KUKA KRL program: MyProgram_126().src

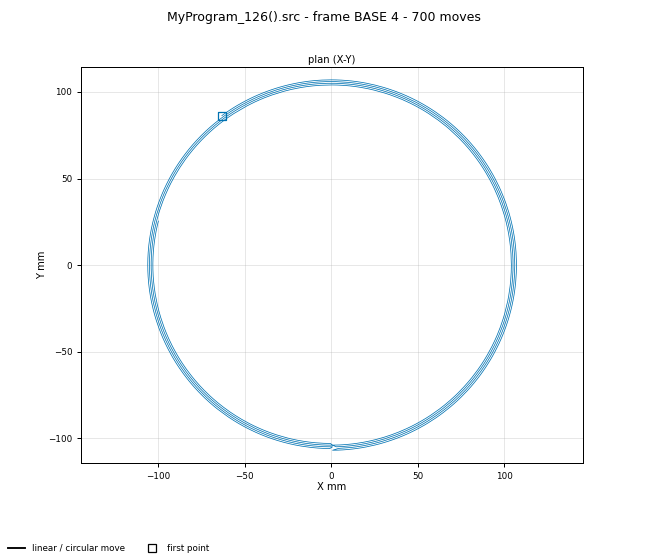
[picture p0: tool path of MyProgram_126().src in frame BASE 4, 700 of 700 moves have a stored position in this frame; points joined in program order, loops and branches not executed]
&ACCESS RVP
&REL 1
&PARAM TEMPLATE = C:\KRC\Roboter\Template\vorgabe
&PARAM EDITMASK = *
DEF MyProgram_126()
; ---- Setting reference (Base) ----
$BASE = BASE_DATA[4]

; --------------------------
; ---- Setting tool (TCP) ----
$TOOL = TOOL_DATA[3]
; --------------------------

$VEL.CP = VEL_APROX_PRINT
Startdeposition()
$VEL.CP = VEL_PRINT
LIN {X -63.1744,Y 86.354,Z 105,A 121.2635,B 24.9294,C -1.9405,E1 24.9063,E2 324.4003} C_DIS
LIN {X -61.0361,Y 87.8784,Z 105,A 119.8304,B 24.9293,C -1.9424,E1 24.9096,E2 325.8339} C_DIS
LIN {X -58.6968,Y 89.4582,Z 105,A 118.2628,B 24.9293,C -1.9432,E1 24.9133,E2 327.4047} C_DIS
LIN {X -56.1298,Y 91.0928,Z 105,A 116.6759,B 24.9289,C -1.9479,E1 24.917,E2 328.9856} C_DIS
LIN {X -53.8773,Y 92.4429,Z 105,A 115.2641,B 24.9287,C -1.9502,E1 24.9204,E2 330.3961} C_DIS
LIN {X -51.5924,Y 93.7373,Z 105,A 113.8527,B 24.9285,C -1.9525,E1 24.9238,E2 331.8062} C_DIS
LIN {X -49.2765,Y 94.9752,Z 105,A 112.4412,B 24.9284,C -1.9546,E1 24.9273,E2 333.2165} C_DIS
LIN {X -46.9308,Y 96.1559,Z 105,A 111.03,B 24.9282,C -1.9567,E1 24.9308,E2 334.6265} C_DIS
LIN {X -44.5569,Y 97.2787,Z 105,A 109.6191,B 24.9281,C -1.9587,E1 24.9344,E2 336.0362} C_DIS
LIN {X -42.1561,Y 98.3428,Z 105,A 108.2082,B 24.9279,C -1.9606,E1 24.938,E2 337.4459} C_DIS
LIN {X -39.73,Y 99.3478,Z 105,A 106.7979,B 24.9278,C -1.9624,E1 24.9416,E2 338.8551} C_DIS
LIN {X -37.2799,Y 100.2929,Z 105,A 105.3874,B 24.9277,C -1.9641,E1 24.9453,E2 340.2644} C_DIS
LIN {X -34.8074,Y 101.1776,Z 105,A 103.9775,B 24.9276,C -1.9657,E1 24.949,E2 341.6733} C_DIS
LIN {X -32.3139,Y 102.0013,Z 105,A 102.5675,B 24.9274,C -1.9672,E1 24.9528,E2 343.0822} C_DIS
LIN {X -29.8009,Y 102.7636,Z 105,A 101.1579,B 24.9274,C -1.9687,E1 24.9566,E2 344.4908} C_DIS
LIN {X -27.27,Y 103.464,Z 105,A 99.7486,B 24.9272,C -1.97,E1 24.9604,E2 345.8991} C_DIS
LIN {X -24.7226,Y 104.1021,Z 105,A 98.1893,B 24.9276,C -1.9655,E1 24.9646,E2 347.4712} C_DIS
LIN {X -21.4758,Y 104.818,Z 105,A 96.576,B 24.927,C -1.9735,E1 24.969,E2 349.0675} C_DIS
LIN {X -18.7569,Y 105.3387,Z 105,A 95.0092,B 24.9271,C -1.9714,E1 24.9733,E2 350.6409} C_DIS
LIN {X -15.6998,Y 105.8394,Z 105,A 93.4091,B 24.9269,C -1.9748,E1 24.9777,E2 352.2345} C_DIS
LIN {X -13.0976,Y 106.1928,Z 105,A 92.001,B 24.9269,C -1.9755,E1 24.9816,E2 353.6417} C_DIS
LIN {X -10.4876,Y 106.4822,Z 105,A 90.5932,B 24.9268,C -1.9762,E1 24.9855,E2 355.0487} C_DIS
LIN {X -7.8712,Y 106.7075,Z 105,A 89.1853,B 24.9268,C -1.9768,E1 24.9894,E2 356.4559} C_DIS
LIN {X -5.2501,Y 106.8686,Z 105,A 87.778,B 24.9267,C -1.9773,E1 24.9933,E2 357.8624} C_DIS
LIN {X -2.6258,Y 106.9652,Z 105,A 86.3708,B 24.9267,C -1.9777,E1 24.9973,E2 359.2689} C_DIS
LIN {X -0.0646,Y 106.9971,Z 105,A 84.9971,B 24.9267,C -1.9779,E1 25.0011,E2 360.6421} C_DIS
LIN {X 2.7297,Y 106.962,Z 105,A 83.3358,B 24.9271,C -1.9716,E1 25.0058,E2 362.318} C_DIS
LIN {X 5.8633,Y 106.8347,Z 105,A 81.8013,B 24.9267,C -1.9774,E1 25.01,E2 363.8383} C_DIS
LIN {X 8.8815,Y 106.6268,Z 105,A 80.1746,B 24.9267,C -1.9771,E1 25.0145,E2 365.465} C_DIS
LIN {X 11.7935,Y 106.3455,Z 105,A 78.6358,B 24.9267,C -1.9779,E1 25.0188,E2 367.0008} C_DIS
LIN {X 14.8232,Y 105.9639,Z 105,A 76.9473,B 24.9268,C -1.9755,E1 25.0235,E2 368.6937} C_DIS
LIN {X 17.6867,Y 105.5235,Z 105,A 75.4509,B 24.9268,C -1.9772,E1 25.0276,E2 370.1846} C_DIS
LIN {X 20.2711,Y 105.0576,Z 105,A 74.0666,B 24.9267,C -1.9775,E1 25.0314,E2 371.5666} C_DIS
LIN {X 22.8432,Y 104.5285,Z 105,A 72.6618,B 24.9267,C -1.9769,E1 25.0352,E2 372.9711} C_DIS
LIN {X 25.3193,Y 103.9565,Z 105,A 71.2816,B 24.9268,C -1.9753,E1 25.039,E2 374.3529} C_DIS
LIN {X 27.9447,Y 103.2818,Z 105,A 69.8529,B 24.9268,C -1.9753,E1 25.0428,E2 375.7794} C_DIS
LIN {X 30.3725,Y 102.594,Z 105,A 68.4576,B 24.927,C -1.9726,E1 25.0466,E2 377.1788} C_DIS
LIN {X 32.9788,Y 101.7862,Z 105,A 67.0452,B 24.927,C -1.9734,E1 25.0504,E2 378.5867} C_DIS
LIN {X 35.4669,Y 100.9462,Z 105,A 65.6414,B 24.927,C -1.9723,E1 25.0541,E2 379.9903} C_DIS
LIN {X 37.9335,Y 100.0454,Z 105,A 64.2171,B 24.9272,C -1.9702,E1 25.0578,E2 381.4165} C_DIS
LIN {X 40.7094,Y 98.9491,Z 105,A 62.6093,B 24.9274,C -1.9682,E1 25.062,E2 383.0255} C_DIS
LIN {X 43.3598,Y 97.8181,Z 105,A 61.0832,B 24.9274,C -1.9672,E1 25.0659,E2 384.5504} C_DIS
LIN {X 45.7473,Y 96.7246,Z 105,A 59.6806,B 24.9276,C -1.9656,E1 25.0694,E2 385.953} C_DIS
LIN {X 48.5601,Y 95.3413,Z 105,A 57.9774,B 24.9278,C -1.9625,E1 25.0737,E2 387.6589} C_DIS
LIN {X 50.9781,Y 94.0705,Z 105,A 56.5274,B 24.9278,C -1.9611,E1 25.0773,E2 389.1083} C_DIS
LIN {X 53.3448,Y 92.7489,Z 105,A 55.1011,B 24.928,C -1.9601,E1 25.0807,E2 390.5327} C_DIS
LIN {X 55.9034,Y 91.2304,Z 105,A 53.5,B 24.9282,C -1.9574,E1 25.0845,E2 392.1353} C_DIS
LIN {X 58.3484,Y 89.6879,Z 105,A 51.97,B 24.9282,C -1.9556,E1 25.0881,E2 393.6644} C_DIS
LIN {X 60.5319,Y 88.229,Z 105,A 50.5686,B 24.9285,C -1.9535,E1 25.0914,E2 395.0661} C_DIS
LIN {X 62.6789,Y 86.7169,Z 105,A 49.1677,B 24.9286,C -1.9513,E1 25.0946,E2 396.4672} C_DIS
LIN {X 64.7784,Y 85.1599,Z 105,A 47.7733,B 24.9288,C -1.9491,E1 25.0977,E2 397.862} C_DIS
LIN {X 66.8584,Y 83.5369,Z 105,A 46.3663,B 24.929,C -1.9467,E1 25.1008,E2 399.2694} C_DIS
LIN {X 68.8883,Y 81.871,Z 105,A 44.9655,B 24.9291,C -1.9442,E1 25.1038,E2 400.6706} C_DIS
LIN {X 70.8768,Y 80.1557,Z 105,A 43.5655,B 24.9293,C -1.9417,E1 25.1067,E2 402.071} C_DIS
LIN {X 72.8226,Y 78.3921,Z 105,A 42.1654,B 24.9295,C -1.9391,E1 25.1096,E2 403.4717} C_DIS
LIN {X 74.7245,Y 76.5814,Z 105,A 40.7655,B 24.9297,C -1.9364,E1 25.1124,E2 404.872} C_DIS
LIN {X 76.5814,Y 74.7245,Z 105,A 39.3658,B 24.9299,C -1.9337,E1 25.1152,E2 406.2723} C_DIS
LIN {X 78.3921,Y 72.8226,Z 105,A 37.8771,B 24.9304,C -1.9271,E1 25.118,E2 407.77} C_DIS
LIN {X 80.5597,Y 70.4142,Z 105,A 36.1898,B 24.9305,C -1.9252,E1 25.1212,E2 409.4543} C_DIS
LIN {X 82.7102,Y 67.8785,Z 105,A 34.4682,B 24.9306,C -1.9234,E1 25.1242,E2 411.1721} C_DIS
LIN {X 84.3511,Y 65.8282,Z 105,A 33.0692,B 24.9309,C -1.9203,E1 25.1267,E2 412.5719} C_DIS
LIN {X 85.9412,Y 63.7383,Z 105,A 31.6706,B 24.9311,C -1.9172,E1 25.129,E2 413.9712} C_DIS
LIN {X 87.4795,Y 61.61,Z 105,A 30.2719,B 24.9313,C -1.914,E1 25.1313,E2 415.3707} C_DIS
LIN {X 88.9651,Y 59.4446,Z 105,A 28.8735,B 24.9316,C -1.9107,E1 25.1335,E2 416.7699} C_DIS
LIN {X 90.3972,Y 57.2434,Z 105,A 27.475,B 24.9318,C -1.9074,E1 25.1356,E2 418.1692} C_DIS
LIN {X 91.7748,Y 55.0077,Z 105,A 25.9012,B 24.9326,C -1.8965,E1 25.1379,E2 419.7607} C_DIS
LIN {X 93.4378,Y 52.1286,Z 105,A 24.3272,B 24.9323,C -1.9005,E1 25.14,E2 421.3171} C_DIS
LIN {X 94.689,Y 49.8199,Z 105,A 22.9293,B 24.9325,C -1.897,E1 25.1419,E2 422.7159} C_DIS
LIN {X 95.8831,Y 47.4811,Z 105,A 21.5111,B 24.9329,C -1.8925,E1 25.1437,E2 424.1371} C_DIS
LIN {X 96.9837,Y 45.1905,Z 105,A 20.138,B 24.9332,C -1.8882,E1 25.1453,E2 425.5132} C_DIS
LIN {X 98.0974,Y 42.7191,Z 105,A 18.7158,B 24.9334,C -1.8852,E1 25.1469,E2 426.9345} C_DIS
LIN {X 99.1163,Y 40.2988,Z 105,A 17.3391,B 24.9336,C -1.8824,E1 25.1484,E2 428.3102} C_DIS
LIN {X 100.0454,Y 37.9335,Z 105,A 15.9456,B 24.934,C -1.877,E1 25.1498,E2 429.7088} C_DIS
LIN {X 100.9462,Y 35.4668,Z 105,A 14.5483,B 24.9342,C -1.8732,E1 25.1511,E2 431.1072} C_DIS
LIN {X 101.8123,Y 32.8982,Z 105,A 13.1473,B 24.9344,C -1.871,E1 25.1523,E2 432.5055} C_DIS
LIN {X 102.5649,Y 30.4709,Z 105,A 11.7541,B 24.9348,C -1.8655,E1 25.1535,E2 433.9037} C_DIS
LIN {X 103.2818,Y 27.9447,Z 105,A 10.357,B 24.935,C -1.8616,E1 25.1545,E2 435.302} C_DIS
LIN {X 103.9859,Y 25.199,Z 105,A 8.8143,B 24.9354,C -1.8558,E1 25.1556,E2 436.8494} C_DIS
LIN {X 104.6775,Y 22.1604,Z 105,A 7.2123,B 24.9356,C -1.8535,E1 25.1565,E2 438.4476} C_DIS
LIN {X 105.1898,Y 19.5848,Z 105,A 5.8156,B 24.9359,C -1.8495,E1 25.1573,E2 439.8456} C_DIS
LIN {X 105.696,Y 16.627,Z 105,A 4.1294,B 24.9365,C -1.841,E1 25.158,E2 441.5418} C_DIS
LIN {X 106.1237,Y 13.6311,Z 105,A 2.534,B 24.9367,C -1.8369,E1 25.1586,E2 443.1374} C_DIS
LIN {X 106.4822,Y 10.4876,Z 105,A 0.9274,B 24.9369,C -1.8353,E1 25.1591,E2 444.7384} C_DIS
LIN {X 106.7394,Y 7.4006,Z 105,A -0.7805,B 24.9374,C -1.8279,E1 25.1595,E2 446.4537} C_DIS
LIN {X 106.8986,Y 4.5519,Z 105,A -2.2374,B 24.9375,C -1.826,E1 25.1597,E2 447.9063} C_DIS
LIN {X 106.9765,Y 2.0118,Z 105,A -3.6153,B 24.9379,C -1.8209,E1 25.1597,E2 449.2881} C_DIS
LIN {X 106.9894,Y -1.313,Z 105,A -5.3568,B 24.9381,C -1.8168,E1 25.1597,E2 451.029} C_DIS
LIN {X 106.8986,Y -4.5519,Z 105,A -7.0801,B 24.9385,C -1.8117,E1 25.1596,E2 452.754} C_DIS
LIN {X 106.749,Y -7.2585,Z 105,A -8.5008,B 24.9387,C -1.8083,E1 25.1594,E2 454.1742} C_DIS
LIN {X 106.5465,Y -9.7916,Z 105,A -9.8935,B 24.9391,C -1.8025,E1 25.159,E2 455.5723} C_DIS
LIN {X 106.2741,Y -12.4035,Z 105,A -11.2899,B 24.9394,C -1.7984,E1 25.1586,E2 456.9701} C_DIS
LIN {X 105.9377,Y -15.0078,Z 105,A -12.6659,B 24.9396,C -1.7951,E1 25.1581,E2 458.3457} C_DIS
LIN {X 105.5375,Y -17.6032,Z 105,A -14.0828,B 24.9399,C -1.7901,E1 25.1575,E2 459.766} C_DIS
LIN {X 104.993,Y -20.6067,Z 105,A -15.7082,B 24.9403,C -1.7853,E1 25.1566,E2 461.3934} C_DIS
LIN {X 104.3976,Y -23.4433,Z 105,A -17.2269,B 24.9405,C -1.7817,E1 25.1557,E2 462.9117} C_DIS
LIN {X 103.7909,Y -25.9983,Z 105,A -18.8086,B 24.9413,C -1.7696,E1 25.1546,E2 464.5128} C_DIS
LIN {X 102.9542,Y -29.1285,Z 105,A -20.3672,B 24.9412,C -1.7718,E1 25.1535,E2 466.0574} C_DIS
LIN {X 102.2083,Y -31.6463,Z 105,A -21.764,B 24.9414,C -1.7677,E1 25.1524,E2 467.4557} C_DIS
LIN {X 101.2929,Y -34.4655,Z 105,A -23.3577,B 24.9418,C -1.7624,E1 25.151,E2 469.0529} C_DIS
LIN {X 100.2929,Y -37.2799,Z 105,A -24.9085,B 24.942,C -1.7595,E1 25.1495,E2 470.6019} C_DIS
LIN {X 99.3478,Y -39.73,Z 105,A -26.3054,B 24.9422,C -1.7556,E1 25.1481,E2 472.0003} C_DIS
LIN {X 98.2923,Y -42.2721,Z 105,A -27.9259,B 24.9429,C -1.7448,E1 25.1463,E2 473.6375} C_DIS
LIN {X 96.9837,Y -45.1905,Z 105,A -29.4507,B 24.9428,C -1.7477,E1 25.1445,E2 475.1471} C_DIS
LIN {X 95.8831,Y -47.4811,Z 105,A -30.8236,B 24.9431,C -1.7431,E1 25.1428,E2 476.5235} C_DIS
LIN {X 94.689,Y -49.8199,Z 105,A -32.2941,B 24.9435,C -1.7361,E1 25.1409,E2 478.0027} C_DIS
LIN {X 93.0971,Y -52.7389,Z 105,A -33.9899,B 24.9436,C -1.7345,E1 25.1387,E2 479.6934} C_DIS
LIN {X 91.7748,Y -55.0077,Z 105,A -35.3873,B 24.9439,C -1.7308,E1 25.1367,E2 481.0924} C_DIS
LIN {X 90.3972,Y -57.2434,Z 105,A -36.785,B 24.9441,C -1.7271,E1 25.1346,E2 482.4917} C_DIS
LIN {X 89.1491,Y -59.1656,Z 105,A -38.0378,B 24.9444,C -1.7226,E1 25.1327,E2 483.7489} C_DIS
LIN {X 87.4795,Y -61.61,Z 105,A -39.5805,B 24.9446,C -1.7199,E1 25.1302,E2 485.2903} C_DIS
LIN {X 85.9412,Y -63.7383,Z 105,A -40.9784,B 24.9448,C -1.7164,E1 25.1279,E2 486.6897} C_DIS
LIN {X 84.3511,Y -65.8282,Z 105,A -42.3762,B 24.945,C -1.713,E1 25.1255,E2 488.089} C_DIS
LIN {X 82.4335,Y -68.2114,Z 105,A -44.057,B 24.9454,C -1.7069,E1 25.1226,E2 489.7765} C_DIS
LIN {X 80.5597,Y -70.4142,Z 105,A -45.5452,B 24.9454,C -1.7054,E1 25.1198,E2 491.2614} C_DIS
LIN {X 78.8074,Y -72.3701,Z 105,A -46.9229,B 24.9456,C -1.703,E1 25.1173,E2 492.6386} C_DIS
LIN {X 77.0076,Y -74.2823,Z 105,A -48.3425,B 24.9459,C -1.699,E1 25.1145,E2 494.0617} C_DIS
LIN {X 75.2217,Y -76.0902,Z 105,A -49.6959,B 24.9461,C -1.6959,E1 25.1119,E2 495.4164} C_DIS
LIN {X 73.1659,Y -78.0693,Z 105,A -51.2769,B 24.9465,C -1.69,E1 25.1086,E2 497.0049} C_DIS
LIN {X 70.8768,Y -80.1557,Z 105,A -52.8664,B 24.9465,C -1.6891,E1 25.1053,E2 498.5904} C_DIS
LIN {X 68.8883,Y -81.871,Z 105,A -54.2659,B 24.9467,C -1.6861,E1 25.1024,E2 499.9913} C_DIS
LIN {X 66.8584,Y -83.5369,Z 105,A -55.6655,B 24.9469,C -1.6833,E1 25.0993,E2 501.3923} C_DIS
LIN {X 64.8233,Y -85.1254,Z 105,A -57.0421,B 24.9471,C -1.6806,E1 25.0963,E2 502.7703} C_DIS
LIN {X 62.6789,Y -86.7169,Z 105,A -58.4649,B 24.9472,C -1.6779,E1 25.0931,E2 504.1944} C_DIS
LIN {X 60.5319,Y -88.229,Z 105,A -59.865,B 24.9474,C -1.6753,E1 25.0899,E2 505.5959} C_DIS
LIN {X 58.3484,Y -89.6879,Z 105,A -61.2652,B 24.9476,C -1.6727,E1 25.0866,E2 506.9974} C_DIS
LIN {X 56.2056,Y -91.0455,Z 105,A -62.6208,B 24.9477,C -1.6703,E1 25.0834,E2 508.3544} C_DIS
LIN {X 53.8773,Y -92.4429,Z 105,A -64.0664,B 24.9479,C -1.6679,E1 25.0799,E2 509.8012} C_DIS
LIN {X 51.0773,Y -94.0167,Z 105,A -65.8081,B 24.9481,C -1.664,E1 25.0756,E2 511.5471} C_DIS
LIN {X 48.6541,Y -95.2932,Z 105,A -67.2779,B 24.9483,C -1.6614,E1 25.072,E2 513.0189} C_DIS
LIN {X 45.7473,Y -96.7246,Z 105,A -68.9703,B 24.9483,C -1.6603,E1 25.0677,E2 514.7094} C_DIS
LIN {X 43.3598,Y -97.8181,Z 105,A -70.3718,B 24.9485,C -1.6584,E1 25.0642,E2 516.1121} C_DIS
LIN {X 40.9462,Y -98.8528,Z 105,A -71.7738,B 24.9485,C -1.6565,E1 25.0606,E2 517.5152} C_DIS
LIN {X 38.0834,Y -99.9886,Z 105,A -73.4838,B 24.9489,C -1.6517,E1 25.0561,E2 519.2328} C_DIS
LIN {X 35.4668,Y -100.9462,Z 105,A -74.9266,B 24.9489,C -1.6517,E1 25.0523,E2 520.6724} C_DIS
LIN {X 32.9788,Y -101.7862,Z 105,A -76.329,B 24.9489,C -1.6502,E1 25.0486,E2 522.076} C_DIS
LIN {X 30.4709,Y -102.5649,Z 105,A -77.7318,B 24.9491,C -1.6487,E1 25.0448,E2 523.4797} C_DIS
LIN {X 27.9447,Y -103.2818,Z 105,A -79.1139,B 24.9491,C -1.6481,E1 25.0411,E2 524.8609} C_DIS
LIN {X 25.4016,Y -103.9364,Z 105,A -80.5378,B 24.9492,C -1.646,E1 25.0373,E2 526.2877} C_DIS
LIN {X 22.7604,Y -104.5466,Z 105,A -81.9658,B 24.9492,C -1.6456,E1 25.0334,E2 527.7148} C_DIS
LIN {X 20.2711,Y -105.0576,Z 105,A -83.3242,B 24.9493,C -1.6445,E1 25.0296,E2 529.0741} C_DIS
LIN {X 17.6032,Y -105.5375,Z 105,A -84.7734,B 24.9493,C -1.6435,E1 25.0257,E2 530.5241} C_DIS
LIN {X 15.0078,Y -105.9377,Z 105,A -86.1568,B 24.9493,C -1.6435,E1 25.0218,E2 531.9064} C_DIS
LIN {X 12.4035,Y -106.2741,Z 105,A -87.6487,B 24.9497,C -1.6391,E1 25.0177,E2 533.4075} C_DIS
LIN {X 9.1801,Y -106.6029,Z 105,A -89.3147,B 24.9495,C -1.6409,E1 25.0131,E2 535.0682} C_DIS
LIN {X 6.5612,Y -106.7961,Z 105,A -90.7196,B 24.9495,C -1.6403,E1 25.0091,E2 536.4738} C_DIS
LIN {X 3.9383,Y -106.925,Z 105,A -92.1248,B 24.9496,C -1.6398,E1 25.0052,E2 537.8798} C_DIS
LIN {X 0.7445,Y -106.9929,Z 105,A -93.5572,B 24.9489,C -1.6506,E1 25.0013,E2 539.2863} C_DIS
Enddeposition()
LIN {X 0.7445,Y -106.9929,Z 105,A -93.5572,B 24.9489,C -1.6506,E1 25.0013,E2 539.2863} C_DIS
Startdeposition()
$VEL.CP = VEL_PRINT
LIN {X 4.2432,Y -105.9303,Z 105,A -91.1652,B 24.9466,C -1.6886,E1 25.0082,E2 536.8049} C_DIS
LIN {X 11.5184,Y -105.3883,Z 105,A -87.286,B 24.9466,C -1.6879,E1 25.019,E2 532.9294} C_DIS
LIN {X 14.8928,Y -104.9636,Z 105,A -85.5122,B 24.9466,C -1.6865,E1 25.0239,E2 531.1604} C_DIS
LIN {X 18.3102,Y -104.4227,Z 105,A -83.5436,B 24.9464,C -1.6919,E1 25.0294,E2 529.1809} C_DIS
LIN {X 21.614,Y -103.7886,Z 105,A -81.7098,B 24.9462,C -1.6942,E1 25.0344,E2 527.3441} C_DIS
LIN {X 25.2421,Y -102.966,Z 105,A -79.8095,B 24.9464,C -1.6916,E1 25.0395,E2 525.4526} C_DIS
LIN {X 29.2068,Y -101.9127,Z 105,A -77.6403,B 24.9464,C -1.692,E1 25.0454,E2 523.2859} C_DIS
LIN {X 33.4613,Y -100.5966,Z 105,A -75.367,B 24.9465,C -1.6893,E1 25.0514,E2 521.0231} C_DIS
LIN {X 36.7427,Y -99.445,Z 105,A -73.2502,B 24.9457,C -1.7016,E1 25.057,E2 518.8815} C_DIS
LIN {X 40.0118,Y -98.1743,Z 105,A -71.0999,B 24.9449,C -1.715,E1 25.0627,E2 516.7045} C_DIS
LIN {X 44.7878,Y -96.0895,Z 105,A -68.6309,B 24.9455,C -1.7047,E1 25.0689,E2 514.2659} C_DIS
LIN {X 47.9345,Y -94.5597,Z 105,A -66.7237,B 24.9453,C -1.7085,E1 25.0736,E2 512.3549} C_DIS
LIN {X 50.6883,Y -93.1121,Z 105,A -65.0728,B 24.9452,C -1.7102,E1 25.0777,E2 510.7048} C_DIS
LIN {X 53.5886,Y -91.4744,Z 105,A -63.1884,B 24.9448,C -1.717,E1 25.0823,E2 508.8099} C_DIS
LIN {X 56.7465,Y -89.5509,Z 105,A -60.551,B 24.9427,C -1.7479,E1 25.0887,E2 506.1079} C_DIS
LIN {X 60.4561,Y -87.0874,Z 105,A -59.1243,B 24.9451,C -1.7111,E1 25.0918,E2 504.7728} C_DIS
LIN {X 62.3319,Y -85.7555,Z 105,A -57.5526,B 24.9441,C -1.7276,E1 25.0954,E2 503.1679} C_DIS
LIN {X 65.1454,Y -83.6393,Z 105,A -55.2936,B 24.9428,C -1.7469,E1 25.1005,E2 500.8715} C_DIS
LIN {X 67.7509,Y -81.5411,Z 105,A -53.8256,B 24.9435,C -1.7364,E1 25.1036,E2 499.4339} C_DIS
LIN {X 71.2226,Y -78.5294,Z 105,A -51.3711,B 24.9432,C -1.7409,E1 25.1087,E2 496.9786} C_DIS
LIN {X 73.9765,Y -75.9404,Z 105,A -49.0824,B 24.9422,C -1.7564,E1 25.1134,E2 494.6629} C_DIS
LIN {X 77.8722,Y -71.9388,Z 105,A -46.2879,B 24.9423,C -1.7543,E1 25.1187,E2 491.8854} C_DIS
LIN {X 80.6502,Y -68.8091,Z 105,A -44.2003,B 24.9424,C -1.7527,E1 25.1225,E2 489.811} C_DIS
LIN {X 82.9488,Y -66.0211,Z 105,A -41.1688,B 24.939,C -1.8046,E1 25.128,E2 486.6711} C_DIS
LIN {X 86.5578,Y -61.2134,Z 105,A -39.015,B 24.9415,C -1.766,E1 25.1313,E2 484.6189} C_DIS
LIN {X 88.488,Y -58.3868,Z 105,A -37.1696,B 24.9412,C -1.771,E1 25.1342,E2 482.7708} C_DIS
LIN {X 90.2848,Y -55.5708,Z 105,A -35.323,B 24.9408,C -1.7779,E1 25.1369,E2 480.9173} C_DIS
LIN {X 91.9633,Y -52.7437,Z 105,A -33.6301,B 24.9406,C -1.7795,E1 25.1393,E2 479.2294} C_DIS
LIN {X 93.6379,Y -49.7113,Z 105,A -31.3081,B 24.939,C -1.8045,E1 25.1424,E2 476.8605} C_DIS
LIN {X 95.2195,Y -46.6118,Z 105,A -29.8969,B 24.94,C -1.7898,E1 25.1441,E2 475.4917} C_DIS
LIN {X 96.6063,Y -43.6622,Z 105,A -28.144,B 24.9396,C -1.7948,E1 25.1462,E2 473.7365} C_DIS
LIN {X 97.9717,Y -40.5096,Z 105,A -25.8965,B 24.9381,C -1.8174,E1 25.1486,E2 471.4479} C_DIS
LIN {X 99.6252,Y -36.2488,Z 105,A -23.8546,B 24.9388,C -1.8065,E1 25.1506,E2 469.4432} C_DIS
LIN {X 100.8782,Y -32.5995,Z 105,A -21.8016,B 24.9385,C -1.8116,E1 25.1524,E2 467.3896} C_DIS
LIN {X 101.8013,Y -29.5968,Z 105,A -20.0833,B 24.9381,C -1.8179,E1 25.1538,E2 465.6664} C_DIS
LIN {X 102.6333,Y -26.5626,Z 105,A -18.3862,B 24.9377,C -1.8232,E1 25.155,E2 463.9665} C_DIS
LIN {X 103.3211,Y -23.7466,Z 105,A -16.6793,B 24.9369,C -1.8343,E1 25.1561,E2 462.2433} C_DIS
LIN {X 104.1668,Y -19.7114,Z 105,A -14.0104,B 24.9351,C -1.8607,E1 25.1576,E2 459.5277} C_DIS
LIN {X 104.8614,Y -15.6062,Z 105,A -11.686,B 24.9344,C -1.8712,E1 25.1585,E2 457.1923} C_DIS
LIN {X 105.4186,Y -11.229,Z 105,A -10.3207,B 24.9369,C -1.8345,E1 25.1589,E2 455.9216} C_DIS
LIN {X 105.8389,Y -6.1102,Z 105,A -6.9313,B 24.9344,C -1.8701,E1 25.1596,E2 452.4683} C_DIS
LIN {X 106.0165,Y 0.0334,Z 105,A -3.8486,B 24.9344,C -1.8704,E1 25.1598,E2 449.4032} C_DIS
LIN {X 105.8544,Y 5.8307,Z 105,A -0.993,B 24.9346,C -1.8685,E1 25.1595,E2 446.5693} C_DIS
LIN {X 105.5637,Y 9.7696,Z 105,A 1.586,B 24.9327,C -1.8946,E1 25.1589,E2 443.9439} C_DIS
LIN {X 105.0602,Y 14.2061,Z 105,A 3.913,B 24.9324,C -1.8985,E1 25.1581,E2 441.6215} C_DIS
LIN {X 104.2828,Y 19.0877,Z 105,A 6.2592,B 24.9328,C -1.8928,E1 25.157,E2 439.3024} C_DIS
LIN {X 103.5964,Y 22.5154,Z 105,A 8.1587,B 24.9324,C -1.8992,E1 25.1559,E2 437.399} C_DIS
LIN {X 102.8849,Y 25.5746,Z 105,A 9.8443,B 24.932,C -1.9039,E1 25.1548,E2 435.7119} C_DIS
LIN {X 102.0776,Y 28.625,Z 105,A 11.5858,B 24.9316,C -1.9107,E1 25.1535,E2 433.9645} C_DIS
LIN {X 101.1882,Y 31.6253,Z 105,A 13.2741,B 24.9312,C -1.9157,E1 25.1521,E2 432.2739} C_DIS
LIN {X 99.5416,Y 36.4778,Z 105,A 15.7427,B 24.9315,C -1.911,E1 25.1499,E2 429.8303} C_DIS
LIN {X 98.6927,Y 38.7156,Z 105,A 17.3099,B 24.9304,C -1.9266,E1 25.1483,E2 428.2351} C_DIS
LIN {X 97.3275,Y 42.0313,Z 105,A 19.5952,B 24.9289,C -1.9471,E1 25.1458,E2 425.9139} C_DIS
LIN {X 95.5625,Y 45.9015,Z 105,A 21.4965,B 24.9297,C -1.9365,E1 25.1436,E2 424.0478} C_DIS
LIN {X 94.2778,Y 48.4862,Z 105,A 23.0894,B 24.9293,C -1.9423,E1 25.1415,E2 422.4497} C_DIS
LIN {X 91.7146,Y 53.1766,Z 105,A 25.8072,B 24.9293,C -1.9429,E1 25.1379,E2 419.7447} C_DIS
LIN {X 90.4763,Y 55.256,Z 105,A 27.291,B 24.9284,C -1.9538,E1 25.1357,E2 418.2427} C_DIS
LIN {X 87.9189,Y 59.2408,Z 105,A 29.6607,B 24.9285,C -1.9524,E1 25.1321,E2 415.8882} C_DIS
LIN {X 86.2759,Y 61.6086,Z 105,A 31.3044,B 24.928,C -1.96,E1 25.1294,E2 414.2345} C_DIS
LIN {X 84.224,Y 64.3866,Z 105,A 33.2447,B 24.9274,C -1.9677,E1 25.1262,E2 412.2854} C_DIS
LIN {X 81.9282,Y 67.2852,Z 105,A 35.2815,B 24.9269,C -1.9741,E1 25.1226,E2 410.2429} C_DIS
LIN {X 79.7117,Y 69.8944,Z 105,A 37.0566,B 24.9269,C -1.9752,E1 25.1194,E2 408.4732} C_DIS
LIN {X 77.1499,Y 72.7121,Z 105,A 39.0092,B 24.9269,C -1.9754,E1 25.1157,E2 406.5289} C_DIS
LIN {X 74.8202,Y 75.1085,Z 105,A 40.942,B 24.9262,C -1.9846,E1 25.1118,E2 404.5825} C_DIS
LIN {X 72.478,Y 77.37,Z 105,A 42.5543,B 24.9263,C -1.9821,E1 25.1086,E2 402.9828} C_DIS
LIN {X 69.6428,Y 79.9315,Z 105,A 44.683,B 24.9258,C -1.9888,E1 25.1042,E2 400.8466} C_DIS
LIN {X 66.8635,Y 82.2705,Z 105,A 46.6285,B 24.9256,C -1.9918,E1 25.1,E2 398.9013} C_DIS
LIN {X 64.5148,Y 84.1252,Z 105,A 48.1661,B 24.9256,C -1.9915,E1 25.0966,E2 397.3703} C_DIS
LIN {X 62.0813,Y 85.9386,Z 105,A 50.5438,B 24.9231,C -2.0251,E1 25.0911,E2 394.9216} C_DIS
LIN {X 58.5419,Y 88.3857,Z 105,A 52.6628,B 24.9235,C -2.0202,E1 25.0862,E2 392.8211} C_DIS
LIN {X 55.4833,Y 90.3382,Z 105,A 54.524,B 24.9235,C -2.019,E1 25.0818,E2 390.9686} C_DIS
LIN {X 51.4922,Y 92.6701,Z 105,A 56.5847,B 24.9247,C -2.0045,E1 25.0769,E2 388.9483} C_DIS
LIN {X 48.5493,Y 94.2456,Z 105,A 58.4238,B 24.9244,C -2.0084,E1 25.0723,E2 387.1053} C_DIS
LIN {X 41.0096,Y 97.7619,Z 105,A 62.8692,B 24.9241,C -2.0114,E1 25.0611,E2 382.6639} C_DIS
LIN {X 37.547,Y 99.1432,Z 105,A 64.6654,B 24.9247,C -2.0046,E1 25.0564,E2 380.8879} C_DIS
LIN {X 35.154,Y 100.0167,Z 105,A 66.337,B 24.9237,C -2.0177,E1 25.0519,E2 379.1885} C_DIS
LIN {X 31.5106,Y 101.2237,Z 105,A 68.4054,B 24.9236,C -2.0191,E1 25.0464,E2 377.1206} C_DIS
LIN {X 27.9048,Y 102.2768,Z 105,A 70.4706,B 24.9233,C -2.022,E1 25.0409,E2 375.0522} C_DIS
LIN {X 24.947,Y 103.038,Z 105,A 72.0675,B 24.9234,C -2.0208,E1 25.0366,E2 373.4605} C_DIS
LIN {X 21.4587,Y 103.8205,Z 105,A 73.9812,B 24.9234,C -2.021,E1 25.0314,E2 371.5488} C_DIS
LIN {X 18.2393,Y 104.4354,Z 105,A 75.8,B 24.9232,C -2.0235,E1 25.0263,E2 369.726} C_DIS
LIN {X 14.6105,Y 105.0037,Z 105,A 77.8461,B 24.923,C -2.0265,E1 25.0207,E2 367.6746} C_DIS
LIN {X 10.1845,Y 105.5254,Z 105,A 80.2913,B 24.9229,C -2.0283,E1 25.0139,E2 365.2268} C_DIS
LIN {X 2.4701,Y 105.9873,Z 105,A 84.2303,B 24.9236,C -2.0187,E1 25.003,E2 361.3119} C_DIS
LIN {X -2.7142,Y 105.9814,Z 105,A 87.6448,B 24.9218,C -2.0422,E1 24.9933,E2 357.8415} C_DIS
LIN {X -6.501,Y 105.8173,Z 105,A 89.2964,B 24.923,C -2.0258,E1 24.9888,E2 356.2284} C_DIS
LIN {X -10.0973,Y 105.5335,Z 105,A 91.2095,B 24.9232,C -2.0234,E1 24.9835,E2 354.32} C_DIS
LIN {X -13.6918,Y 105.127,Z 105,A 93.0574,B 24.9236,C -2.0181,E1 24.9784,E2 352.4834} C_DIS
LIN {X -17.0094,Y 104.6425,Z 105,A 94.9457,B 24.9236,C -2.0198,E1 24.9732,E2 350.5894} C_DIS
LIN {X -21.8937,Y 103.7312,Z 105,A 97.706,B 24.9234,C -2.0205,E1 24.9656,E2 347.8244} C_DIS
LIN {X -25.6118,Y 102.8758,Z 105,A 99.7205,B 24.9237,C -2.0168,E1 24.9601,E2 345.816} C_DIS
LIN {X -28.8756,Y 102.0066,Z 105,A 101.8687,B 24.9229,C -2.0273,E1 24.9543,E2 343.6394} C_DIS
LIN {X -32.0493,Y 101.0562,Z 105,A 103.3129,B 24.9241,C -2.0119,E1 24.9505,E2 342.2294} C_DIS
LIN {X -37.4357,Y 99.1853,Z 105,A 106.7138,B 24.9235,C -2.0202,E1 24.9415,E2 338.8018} C_DIS
LIN {X -42.3702,Y 97.1798,Z 105,A 109.0023,B 24.9255,C -1.9936,E1 24.9358,E2 336.5714} C_DIS
LIN {X -44.7455,Y 96.1092,Z 105,A 110.7231,B 24.9248,C -2.0033,E1 24.9313,E2 334.8232} C_DIS
LIN {X -48.3375,Y 94.3538,Z 105,A 112.8755,B 24.925,C -1.9995,E1 24.926,E2 332.6743} C_DIS
LIN {X -51.7657,Y 92.5174,Z 105,A 114.9908,B 24.9253,C -1.9964,E1 24.9208,E2 330.5603} C_DIS
LIN {X -55.8642,Y 90.1025,Z 105,A 117.5529,B 24.9256,C -1.9913,E1 24.9147,E2 328.0024} C_DIS
LIN {X -58.4945,Y 88.417,Z 105,A 119.2381,B 24.9259,C -1.988,E1 24.9107,E2 326.3198} C_DIS
LIN {X -61.5132,Y 86.3439,Z 105,A 121.2617,B 24.9261,C -1.9856,E1 24.9061,E2 324.2947} C_DIS
LIN {X -64.6419,Y 84.0273,Z 105,A 123.3147,B 24.9265,C -1.9793,E1 24.9015,E2 322.2494} C_DIS
LIN {X -67.5086,Y 81.7425,Z 105,A 125.3436,B 24.9267,C -1.9768,E1 24.8971,E2 320.219} C_DIS
LIN {X -70.2018,Y 79.4433,Z 105,A 127.3111,B 24.9269,C -1.9744,E1 24.893,E2 318.2494} C_DIS
LIN {X -72.7237,Y 77.139,Z 105,A 129.0694,B 24.9275,C -1.9668,E1 24.8894,E2 316.5019} C_DIS
LIN {X -75.1228,Y 74.8057,Z 105,A 130.9659,B 24.9275,C -1.9657,E1 24.8856,E2 314.6001} C_DIS
LIN {X -77.7345,Y 72.0888,Z 105,A 133.0415,B 24.9278,C -1.9621,E1 24.8816,E2 312.5242} C_DIS
LIN {X -80.0874,Y 69.4643,Z 105,A 134.8544,B 24.9284,C -1.9538,E1 24.8783,E2 310.7227} C_DIS
LIN {X -82.3312,Y 66.7886,Z 105,A 136.7709,B 24.9287,C -1.95,E1 24.8749,E2 308.8066} C_DIS
LIN {X -84.3667,Y 64.2005,Z 105,A 138.6022,B 24.9289,C -1.9471,E1 24.8718,E2 306.9734} C_DIS
LIN {X -86.336,Y 61.5244,Z 105,A 140.34,B 24.9294,C -1.9401,E1 24.869,E2 305.2438} C_DIS
LIN {X -88.2257,Y 58.7846,Z 105,A 142.3342,B 24.9293,C -1.9422,E1 24.8658,E2 303.2346} C_DIS
LIN {X -90.1623,Y 55.7684,Z 105,A 144.1809,B 24.9299,C -1.9334,E1 24.8631,E2 301.3996} C_DIS
LIN {X -91.9533,Y 52.7612,Z 105,A 146.0153,B 24.9305,C -1.9259,E1 24.8605,E2 299.5736} C_DIS
LIN {X -93.5857,Y 49.8103,Z 105,A 147.9236,B 24.9306,C -1.9236,E1 24.858,E2 297.6605} C_DIS
LIN {X -95.2095,Y 46.6321,Z 105,A 150.0117,B 24.9306,C -1.9237,E1 24.8554,E2 295.5611} C_DIS
LIN {X -96.6686,Y 43.5239,Z 105,A 151.6621,B 24.9316,C -1.9106,E1 24.8535,E2 293.9329} C_DIS
LIN {X -97.7873,Y 40.9494,Z 105,A 153.8355,B 24.9302,C -1.93,E1 24.8511,E2 291.7011} C_DIS
LIN {X -99.3389,Y 37.0293,Z 105,A 155.3377,B 24.9327,C -1.8946,E1 24.8497,E2 290.275} C_DIS
LIN {X -100.6127,Y 33.4135,Z 105,A 157.4731,B 24.933,C -1.8904,E1 24.8477,E2 288.1373} C_DIS
LIN {X -101.4354,Y 30.8279,Z 105,A 159.1617,B 24.9328,C -1.8939,E1 24.8463,E2 286.4308} C_DIS
LIN {X -102.6546,Y 26.4798,Z 105,A 161.2016,B 24.9343,C -1.8716,E1 24.8448,E2 284.4321} C_DIS
LIN {X -103.2302,Y 24.1401,Z 105,A 162.8256,B 24.9338,C -1.8791,E1 24.8437,E2 282.7808} C_DIS
LIN {X -103.9101,Y 21.0221,Z 105,A 164.5111,B 24.9343,C -1.8722,E1 24.8428,E2 281.1019} C_DIS
LIN {X -104.4819,Y 17.9697,Z 105,A 166.2878,B 24.9344,C -1.8703,E1 24.8419,E2 279.3191} C_DIS
LIN {X -105.025,Y 14.46,Z 105,A 168.2769,B 24.9347,C -1.8667,E1 24.8411,E2 277.3268} C_DIS
LIN {X -105.4069,Y 11.3411,Z 105,A 169.9606,B 24.9351,C -1.8607,E1 24.8406,E2 275.6473} C_DIS
LIN {X -105.7558,Y 7.4113,Z 105,A 172.0568,B 24.9357,C -1.8525,E1 24.8401,E2 273.5581} C_DIS
LIN {X -105.9439,Y 3.9277,Z 105,A 174.0791,B 24.9357,C -1.8513,E1 24.8398,E2 271.5263} C_DIS
LIN {X -106.0161,Y 0.1301,Z 105,A 176.1208,B 24.9362,C -1.8443,E1 24.8398,E2 269.4892} C_DIS
LIN {X -105.9596,Y -3.4251,Z 105,A 177.9207,B 24.937,C -1.8337,E1 24.8399,E2 267.7036} C_DIS
LIN {X -105.8041,Y -6.6965,Z 105,A 179.7887,B 24.9371,C -1.8316,E1 24.8402,E2 265.8295} C_DIS
LIN {X -105.5063,Y -10.3915,Z 105,A -178.1116,B 24.9373,C -1.8287,E1 24.8407,E2 263.7242} C_DIS
LIN {X -105.0693,Y -14.1372,Z 105,A -176.0707,B 24.9378,C -1.8223,E1 24.8415,E2 261.6862} C_DIS
LIN {X -104.5114,Y -17.7938,Z 105,A -174.2122,B 24.9385,C -1.8109,E1 24.8423,E2 259.8439} C_DIS
LIN {X -103.9049,Y -21.0474,Z 105,A -172.4126,B 24.9389,C -1.8057,E1 24.8432,E2 258.0461} C_DIS
LIN {X -102.9185,Y -25.4366,Z 105,A -169.999,B 24.9394,C -1.7975,E1 24.8448,E2 255.6378} C_DIS
LIN {X -102.0852,Y -28.5982,Z 105,A -168.1005,B 24.9394,C -1.7969,E1 24.8462,E2 253.7297} C_DIS
LIN {X -101.1198,Y -31.8458,Z 105,A -166.3011,B 24.9399,C -1.7902,E1 24.8476,E2 251.9359} C_DIS
LIN {X -99.5148,Y -36.5514,Z 105,A -163.697,B 24.9407,C -1.7792,E1 24.85,E2 249.3434} C_DIS
LIN {X -98.3741,Y -39.521,Z 105,A -161.8413,B 24.9407,C -1.7792,E1 24.8519,E2 247.4774} C_DIS
LIN {X -97.1393,Y -42.4631,Z 105,A -160.1503,B 24.9411,C -1.773,E1 24.8538,E2 245.7917} C_DIS
LIN {X -95.7001,Y -45.6151,Z 105,A -158.2002,B 24.9412,C -1.7705,E1 24.8561,E2 243.8368} C_DIS
LIN {X -94.2829,Y -48.4763,Z 105,A -156.5008,B 24.9416,C -1.7647,E1 24.8582,E2 242.142} C_DIS
LIN {X -92.5103,Y -51.7784,Z 105,A -154.5337,B 24.9421,C -1.7571,E1 24.8608,E2 240.1829} C_DIS
LIN {X -91.2656,Y -53.942,Z 105,A -153.1411,B 24.9423,C -1.7551,E1 24.8628,E2 238.7879} C_DIS
LIN {X -89.5134,Y -56.8049,Z 105,A -151.2748,B 24.9425,C -1.7522,E1 24.8656,E2 236.9188} C_DIS
LIN {X -87.7139,Y -59.5435,Z 105,A -149.611,B 24.943,C -1.7437,E1 24.8681,E2 235.2669} C_DIS
LIN {X -85.363,Y -62.868,Z 105,A -147.3772,B 24.9433,C -1.7394,E1 24.8718,E2 233.0324} C_DIS
LIN {X -83.0887,Y -65.844,Z 105,A -145.4212,B 24.9438,C -1.732,E1 24.8751,E2 231.0849} C_DIS
LIN {X -81.5378,Y -67.7549,Z 105,A -143.4987,B 24.9425,C -1.7512,E1 24.8786,E2 229.1079} C_DIS
LIN {X -79.2784,Y -70.3866,Z 105,A -142.2449,B 24.9443,C -1.7235,E1 24.8808,E2 227.9143} C_DIS
LIN {X -76.4535,Y -73.4441,Z 105,A -139.7722,B 24.9441,C -1.7269,E1 24.8856,E2 225.4226} C_DIS
LIN {X -73.3009,Y -76.5915,Z 105,A -137.653,B 24.9451,C -1.7109,E1 24.8897,E2 223.3326} C_DIS
LIN {X -70.2272,Y -79.4211,Z 105,A -134.9679,B 24.9444,C -1.7226,E1 24.8954,E2 220.609} C_DIS
LIN {X -67.5881,Y -81.6765,Z 105,A -133.265,B 24.945,C -1.7124,E1 24.899,E2 218.9237} C_DIS
LIN {X -65.4607,Y -83.3916,Z 105,A -131.7574,B 24.9451,C -1.7109,E1 24.9023,E2 217.4142} C_DIS
LIN {X -59.526,Y -87.7257,Z 105,A -127.7199,B 24.9454,C -1.7066,E1 24.9115,E2 213.3728} C_DIS
LIN {X -56.315,Y -89.8209,Z 105,A -125.7147,B 24.9458,C -1.7008,E1 24.9161,E2 211.375} C_DIS
LIN {X -53.3918,Y -91.5908,Z 105,A -123.7501,B 24.9457,C -1.7026,E1 24.9209,E2 209.4001} C_DIS
LIN {X -50.2712,Y -93.3384,Z 105,A -121.4452,B 24.9449,C -1.7145,E1 24.9266,E2 207.0604} C_DIS
LIN {X -47.2609,Y -94.8978,Z 105,A -119.6759,B 24.9452,C -1.7098,E1 24.931,E2 205.2977} C_DIS
LIN {X -43.5067,Y -96.6763,Z 105,A -117.92,B 24.9466,C -1.6881,E1 24.9354,E2 203.5888} C_DIS
LIN {X -40.4374,Y -98.0011,Z 105,A -115.8915,B 24.9462,C -1.6949,E1 24.9406,E2 201.5397} C_DIS
LIN {X -36.8576,Y -99.4031,Z 105,A -113.7919,B 24.9462,C -1.6938,E1 24.9461,E2 199.4382} C_DIS
LIN {X -33.6829,Y -100.5219,Z 105,A -112.1493,B 24.9468,C -1.6853,E1 24.9504,E2 197.8125} C_DIS
LIN {X -31.0386,Y -101.37,Z 105,A -110.4985,B 24.9465,C -1.6901,E1 24.9548,E2 196.1475} C_DIS
LIN {X -27.6516,Y -102.3452,Z 105,A -108.6515,B 24.9467,C -1.6866,E1 24.9598,E2 194.3059} C_DIS
LIN {X -24.114,Y -103.2363,Z 105,A -106.6615,B 24.9467,C -1.6863,E1 24.9652,E2 192.314} C_DIS
LIN {X -20.7561,Y -103.9647,Z 105,A -104.7937,B 24.9467,C -1.6859,E1 24.9703,E2 190.4448} C_DIS
LIN {X -17.3466,Y -104.5861,Z 105,A -102.9477,B 24.9468,C -1.6842,E1 24.9754,E2 188.601} C_DIS
LIN {X -11.4572,Y -105.3947,Z 105,A -99.6767,B 24.9468,C -1.6859,E1 24.9845,E2 185.3236} C_DIS
LIN {X -7.6455,Y -105.7399,Z 105,A -97.837,B 24.9473,C -1.6767,E1 24.9895,E2 183.505} C_DIS
LIN {X -4.8052,Y -105.9062,Z 105,A -95.5691,B 24.9454,C -1.7063,E1 24.9961,E2 181.1663} C_DIS
LIN {X -0.8568,Y -106.0116,Z 105,A -94.038,B 24.947,C -1.6822,E1 25.0002,E2 179.6922} C_DIS
LIN {X -0.8568,Y -106.0116,Z 105,A -94.038,B 24.947,C -1.6822,E1 25.0002,E2 179.6922} C_DIS
Enddeposition()
LIN {X 0.7254,Y -105.0307,Z 105,A -94.1271,B 24.9482,C -1.6619,E1 24.9998,E2 179.8294} C_DIS
Startdeposition()
$VEL.CP = VEL_PRINT
LIN {X -4.7295,Y -104.9279,Z 105,A -96.5021,B 24.9468,C -1.6851,E1 24.9933,E2 182.1497} C_DIS
LIN {X -10.4176,Y -104.5176,Z 105,A -100.1753,B 24.9482,C -1.663,E1 24.9829,E2 185.8769} C_DIS
LIN {X -14.3403,Y -104.0516,Z 105,A -102.2468,B 24.9479,C -1.6667,E1 24.9772,E2 187.9412} C_DIS
LIN {X -17.3669,Y -103.5885,Z 105,A -103.9207,B 24.9479,C -1.667,E1 24.9726,E2 189.6158} C_DIS
LIN {X -21.0855,Y -102.896,Z 105,A -105.973,B 24.9479,C -1.6682,E1 24.967,E2 191.6674} C_DIS
LIN {X -24.6294,Y -102.1061,Z 105,A -107.7271,B 24.9472,C -1.678,E1 24.9623,E2 193.4007} C_DIS
LIN {X -27.3585,Y -101.4086,Z 105,A -109.4061,B 24.9475,C -1.6734,E1 24.9577,E2 195.0931} C_DIS
LIN {X -31.6107,Y -100.166,Z 105,A -111.9551,B 24.9477,C -1.67,E1 24.9508,E2 197.6544} C_DIS
LIN {X -34.9092,Y -99.0634,Z 105,A -113.8298,B 24.9476,C -1.6724,E1 24.9459,E2 199.5269} C_DIS
LIN {X -38.1118,Y -97.8763,Z 105,A -115.9967,B 24.9482,C -1.6626,E1 24.9402,E2 201.7216} C_DIS
LIN {X -42.3579,Y -96.1154,Z 105,A -118.2024,B 24.9473,C -1.6767,E1 24.9346,E2 203.899} C_DIS
LIN {X -46.2348,Y -94.3119,Z 105,A -121.0369,B 24.9483,C -1.6606,E1 24.9273,E2 206.7791} C_DIS
LIN {X -49.5124,Y -92.6343,Z 105,A -122.6367,B 24.9472,C -1.6785,E1 24.9235,E2 208.3407} C_DIS
LIN {X -52.9062,Y -90.7387,Z 105,A -124.7308,B 24.947,C -1.6825,E1 24.9184,E2 210.4316} C_DIS
LIN {X -55.2182,Y -89.3498,Z 105,A -126.254,B 24.947,C -1.6827,E1 24.9148,E2 211.9589} C_DIS
LIN {X -58.347,Y -87.3396,Z 105,A -128.0955,B 24.9463,C -1.6929,E1 24.9105,E2 213.7822} C_DIS
LIN {X -61.0574,Y -85.4645,Z 105,A -130.3652,B 24.9472,C -1.6784,E1 24.9052,E2 216.0942} C_DIS
LIN {X -63.6462,Y -83.5565,Z 105,A -131.8418,B 24.9464,C -1.6918,E1 24.902,E2 217.5443} C_DIS
LIN {X -66.8787,Y -80.9909,Z 105,A -133.7706,B 24.9453,C -1.7079,E1 24.8979,E2 219.4419} C_DIS
LIN {X -69.5777,Y -78.6864,Z 105,A -136.0479,B 24.9459,C -1.699,E1 24.893,E2 221.7493} C_DIS
LIN {X -72.3177,Y -76.1747,Z 105,A -138.8233,B 24.9474,C -1.6759,E1 24.8872,E2 224.5911} C_DIS
LIN {X -75.7798,Y -72.7301,Z 105,A -141.1405,B 24.9462,C -1.6942,E1 24.8828,E2 226.8747} C_DIS
LIN {X -78.1507,Y -70.176,Z 105,A -143.0594,B 24.946,C -1.6979,E1 24.8792,E2 228.7935} C_DIS
LIN {X -80.4946,Y -67.476,Z 105,A -144.6089,B 24.9448,C -1.7169,E1 24.8765,E2 230.3047} C_DIS
LIN {X -82.2597,Y -65.3114,Z 105,A -146.2506,B 24.9448,C -1.7163,E1 24.8736,E2 231.9556} C_DIS
LIN {X -84.0725,Y -62.9605,Z 105,A -148.2418,B 24.9454,C -1.7068,E1 24.8702,E2 233.9789} C_DIS
LIN {X -86.2766,Y -59.9044,Z 105,A -149.7831,B 24.9439,C -1.7305,E1 24.8678,E2 235.4714} C_DIS
LIN {X -88.2948,Y -56.888,Z 105,A -151.7887,B 24.9436,C -1.7347,E1 24.8647,E2 237.4771} C_DIS
LIN {X -90.3011,Y -53.6466,Z 105,A -153.8463,B 24.9432,C -1.741,E1 24.8618,E2 239.5303} C_DIS
LIN {X -92.268,Y -50.1878,Z 105,A -156.029,B 24.9428,C -1.7464,E1 24.8588,E2 241.7114} C_DIS
LIN {X -93.6229,Y -47.6129,Z 105,A -157.9288,B 24.9433,C -1.7396,E1 24.8563,E2 243.6376} C_DIS
LIN {X -95.7044,Y -43.2768,Z 105,A -160.3093,B 24.9422,C -1.7557,E1 24.8535,E2 245.9927} C_DIS
LIN {X -97.1627,Y -39.896,Z 105,A -162.2934,B 24.9418,C -1.7624,E1 24.8514,E2 247.9719} C_DIS
LIN {X -98.3339,Y -36.9151,Z 105,A -163.9484,B 24.9412,C -1.7708,E1 24.8497,E2 249.6161} C_DIS
LIN {X -99.9201,Y -32.3752,Z 105,A -167.2466,B 24.9423,C -1.7547,E1 24.8468,E2 252.9715} C_DIS
LIN {X -101.0342,Y -28.7102,Z 105,A -168.7124,B 24.9404,C -1.7832,E1 24.8457,E2 254.3779} C_DIS
LIN {X -102.6788,Y -22.1204,Z 105,A -172.3656,B 24.9395,C -1.7964,E1 24.8433,E2 258.021} C_DIS
LIN {X -103.3321,Y -18.8343,Z 105,A -174.3601,B 24.9395,C -1.7962,E1 24.8422,E2 260.0278} C_DIS
LIN {X -103.8765,Y -15.5597,Z 105,A -176.2436,B 24.9393,C -1.7993,E1 24.8414,E2 261.9151} C_DIS
LIN {X -104.341,Y -12.049,Z 105,A -178.1146,B 24.9388,C -1.8076,E1 24.8407,E2 263.7774} C_DIS
LIN {X -104.6913,Y -8.4807,Z 105,A 179.932,B 24.9383,C -1.8139,E1 24.8402,E2 265.7275} C_DIS
LIN {X -104.9089,Y -5.1671,Z 105,A 177.9845,B 24.9383,C -1.8149,E1 24.8399,E2 267.6844} C_DIS
LIN {X -105.0198,Y -1.7481,Z 105,A 176.1141,B 24.9379,C -1.8208,E1 24.8398,E2 269.552} C_DIS
LIN {X -105.0153,Y 1.9946,Z 105,A 174.1502,B 24.9372,C -1.8301,E1 24.8398,E2 271.5055} C_DIS
LIN {X -104.8863,Y 5.576,Z 105,A 172.1436,B 24.9369,C -1.8346,E1 24.8401,E2 273.5134} C_DIS
LIN {X -104.6338,Y 9.1748,Z 105,A 170.1274,B 24.9366,C -1.8393,E1 24.8405,E2 275.5306} C_DIS
LIN {X -104.3421,Y 12.0396,Z 105,A 168.1315,B 24.9373,C -1.8294,E1 24.8412,E2 277.562} C_DIS
LIN {X -103.8756,Y 15.5656,Z 105,A 166.6596,B 24.9357,C -1.8521,E1 24.8417,E2 278.9886} C_DIS
LIN {X -103.3697,Y 18.6248,Z 105,A 164.8978,B 24.9355,C -1.8551,E1 24.8426,E2 280.7538} C_DIS
LIN {X -102.6726,Y 22.1492,Z 105,A 162.9596,B 24.935,C -1.8621,E1 24.8437,E2 282.6866} C_DIS
LIN {X -101.8452,Y 25.6895,Z 105,A 160.455,B 24.9358,C -1.8501,E1 24.8454,E2 285.2345} C_DIS
LIN {X -100.8694,Y 29.2902,Z 105,A 159.0293,B 24.9339,C -1.8779,E1 24.8464,E2 286.602} C_DIS
LIN {X -98.5596,Y 36.3085,Z 105,A 154.7414,B 24.9336,C -1.8814,E1 24.8503,E2 290.9061} C_DIS
LIN {X -96.9603,Y 40.3866,Z 105,A 152.6505,B 24.9324,C -1.8993,E1 24.8524,E2 292.966} C_DIS
LIN {X -95.519,Y 43.6881,Z 105,A 150.5859,B 24.9322,C -1.9017,E1 24.8547,E2 295.0363} C_DIS
LIN {X -92.9666,Y 48.8815,Z 105,A 147.2828,B 24.9319,C -1.9059,E1 24.8589,E2 298.3471} C_DIS
LIN {X -91.1875,Y 52.1256,Z 105,A 145.2472,B 24.9315,C -1.9112,E1 24.8616,E2 300.3809} C_DIS
LIN {X -89.3237,Y 55.2601,Z 105,A 142.9684,B 24.9319,C -1.9066,E1 24.865,E2 302.6822} C_DIS
LIN {X -86.4321,Y 59.6807,Z 105,A 140.379,B 24.9305,C -1.925,E1 24.8689,E2 305.2406} C_DIS
LIN {X -84.5175,Y 62.3629,Z 105,A 138.4711,B 24.9305,C -1.926,E1 24.8721,E2 307.1555} C_DIS
LIN {X -82.4001,Y 65.1338,Z 105,A 136.6315,B 24.9299,C -1.9333,E1 24.8752,E2 308.9863} C_DIS
LIN {X -80.0266,Y 68.029,Z 105,A 134.5736,B 24.9296,C -1.9381,E1 24.8789,E2 311.0424} C_DIS
LIN {X -77.551,Y 70.8384,Z 105,A 132.5323,B 24.9292,C -1.9433,E1 24.8827,E2 313.0803} C_DIS
LIN {X -75.0839,Y 73.4497,Z 105,A 130.4865,B 24.9291,C -1.945,E1 24.8867,E2 315.1309} C_DIS
LIN {X -72.5816,Y 75.9229,Z 105,A 128.543,B 24.9288,C -1.9487,E1 24.8906,E2 317.0736} C_DIS
LIN {X -69.9088,Y 78.39,Z 105,A 126.5707,B 24.9284,C -1.9538,E1 24.8946,E2 319.0418} C_DIS
LIN {X -67.1388,Y 80.7748,Z 105,A 124.6271,B 24.928,C -1.96,E1 24.8988,E2 320.978} C_DIS
LIN {X -64.239,Y 83.0997,Z 105,A 122.6283,B 24.9276,C -1.9654,E1 24.9031,E2 322.9713} C_DIS
LIN {X -61.5572,Y 85.1074,Z 105,A 120.6815,B 24.9276,C -1.9649,E1 24.9075,E2 324.9264} C_DIS
LIN {X -58.6073,Y 87.1636,Z 105,A 118.702,B 24.9274,C -1.9681,E1 24.9121,E2 326.9048} C_DIS
LIN {X -56.1255,Y 88.7831,Z 105,A 116.4266,B 24.9289,C -1.9473,E1 24.9176,E2 329.237} C_DIS
LIN {X -52.2205,Y 91.133,Z 105,A 114.6384,B 24.9267,C -1.9771,E1 24.9218,E2 330.9596} C_DIS
LIN {X -48.8318,Y 92.9928,Z 105,A 112.5298,B 24.9264,C -1.9807,E1 24.9269,E2 333.0656} C_DIS
LIN {X -45.5338,Y 94.6512,Z 105,A 110.6815,B 24.9257,C -1.99,E1 24.9315,E2 334.8966} C_DIS
LIN {X -40.9482,Y 96.7236,Z 105,A 107.7523,B 24.926,C -1.9873,E1 24.939,E2 337.8394} C_DIS
LIN {X -34.1066,Y 99.3442,Z 105,A 103.9011,B 24.9252,C -1.9979,E1 24.9491,E2 341.6733} C_DIS
LIN {X -28.301,Y 101.1502,Z 105,A 100.4044,B 24.9254,C -1.9949,E1 24.9584,E2 345.1832} C_DIS
LIN {X -24.9418,Y 102.0299,Z 105,A 98.8026,B 24.9244,C -2.0077,E1 24.9627,E2 346.7568} C_DIS
LIN {X -22.3701,Y 102.6244,Z 105,A 96.5858,B 24.9265,C -1.9799,E1 24.9689,E2 349.0425} C_DIS
LIN {X -18.6924,Y 103.3576,Z 105,A 95.0657,B 24.9249,C -2.0012,E1 24.973,E2 350.5136} C_DIS
LIN {X -14.997,Y 103.9583,Z 105,A 93.0116,B 24.9249,C -2.0021,E1 24.9786,E2 352.5673} C_DIS
LIN {X -11.3998,Y 104.4148,Z 105,A 91.0251,B 24.9248,C -2.0029,E1 24.9841,E2 354.5532} C_DIS
LIN {X -8.2261,Y 104.7117,Z 105,A 89.3155,B 24.9246,C -2.0049,E1 24.9889,E2 356.259} C_DIS
LIN {X -2.3302,Y 105.0082,Z 105,A 85.8128,B 24.9254,C -1.9952,E1 24.9987,E2 359.7854} C_DIS
LIN {X 1.8964,Y 105.0171,Z 105,A 84.0184,B 24.9239,C -2.0152,E1 25.0036,E2 361.5323} C_DIS
LIN {X 4.5686,Y 104.9348,Z 105,A 81.9614,B 24.9256,C -1.9923,E1 25.0095,E2 363.643} C_DIS
LIN {X 9.5603,Y 104.5982,Z 105,A 79.5811,B 24.9246,C -2.0055,E1 25.016,E2 365.9906} C_DIS
LIN {X 13.0454,Y 104.2219,Z 105,A 77.6756,B 24.9246,C -2.0055,E1 25.0213,E2 367.895} C_DIS
LIN {X 16.0391,Y 103.8024,Z 105,A 76.0336,B 24.9246,C -2.0053,E1 25.0258,E2 369.5359} C_DIS
LIN {X 19.5755,Y 103.1943,Z 105,A 74.0453,B 24.9247,C -2.0033,E1 25.0313,E2 371.5266} C_DIS
LIN {X 22.2184,Y 102.6575,Z 105,A 72.5358,B 24.9249,C -2.0011,E1 25.0354,E2 373.0394} C_DIS
LIN {X 25.3976,Y 101.9187,Z 105,A 70.394,B 24.926,C -1.986,E1 25.0413,E2 375.214} C_DIS
LIN {X 28.5439,Y 101.0813,Z 105,A 69.0432,B 24.9249,C -2.0014,E1 25.0449,E2 376.5259} C_DIS
LIN {X 32.104,Y 100.0079,Z 105,A 67.0355,B 24.9249,C -2.0007,E1 25.0502,E2 378.5318} C_DIS
LIN {X 35.2858,Y 98.9312,Z 105,A 64.83,B 24.9262,C -1.9844,E1 25.0561,E2 380.7715} C_DIS
LIN {X 39.5502,Y 97.3035,Z 105,A 62.7965,B 24.925,C -1.9999,E1 25.0613,E2 382.7636} C_DIS
LIN {X 42.9646,Y 95.845,Z 105,A 60.2024,B 24.9269,C -1.9751,E1 25.0681,E2 385.41} C_DIS
LIN {X 46.2403,Y 94.3092,Z 105,A 58.7067,B 24.9256,C -1.9917,E1 25.0717,E2 386.8628} C_DIS
LIN {X 49.7905,Y 92.4835,Z 105,A 56.4812,B 24.926,C -1.9869,E1 25.0772,E2 389.0933} C_DIS
LIN {X 53.401,Y 90.4462,Z 105,A 54.2691,B 24.926,C -1.9856,E1 25.0826,E2 391.3017} C_DIS
LIN {X 55.8106,Y 88.9797,Z 105,A 52.5896,B 24.9267,C -1.9776,E1 25.0866,E2 392.9949} C_DIS
LIN {X 61.3175,Y 85.279,Z 105,A 49.2148,B 24.9264,C -1.9814,E1 25.0943,E2 396.3491} C_DIS
LIN {X 64.5627,Y 82.8503,Z 105,A 47.0354,B 24.9266,C -1.9787,E1 25.0992,E2 398.527} C_DIS
LIN {X 67.5451,Y 80.4372,Z 105,A 44.7815,B 24.9274,C -1.9682,E1 25.1041,E2 400.7971} C_DIS
LIN {X 72.1376,Y 76.3441,Z 105,A 41.4337,B 24.9278,C -1.9618,E1 25.111,E2 404.1467} C_DIS
LIN {X 74.775,Y 73.7624,Z 105,A 39.5248,B 24.9278,C -1.9618,E1 25.1147,E2 406.0476} C_DIS
LIN {X 78.3693,Y 69.9319,Z 105,A 36.6286,B 24.9284,C -1.9541,E1 25.1202,E2 408.9492} C_DIS
LIN {X 81.4319,Y 66.3408,Z 105,A 34.0539,B 24.9289,C -1.948,E1 25.1249,E2 411.5264} C_DIS
LIN {X 83.0923,Y 64.2486,Z 105,A 32.468,B 24.9295,C -1.9392,E1 25.1276,E2 413.1257} C_DIS
LIN {X 85.429,Y 61.1072,Z 105,A 30.5297,B 24.9293,C -1.942,E1 25.1308,E2 415.048} C_DIS
LIN {X 86.8727,Y 59.0369,Z 105,A 28.7158,B 24.9309,C -1.9204,E1 25.1337,E2 416.9038} C_DIS
LIN {X 88.7945,Y 56.1071,Z 105,A 27.3374,B 24.9296,C -1.9375,E1 25.1357,E2 418.2351} C_DIS
LIN {X 92.4326,Y 49.8843,Z 105,A 23.2729,B 24.9308,C -1.9213,E1 25.1414,E2 422.3166} C_DIS
LIN {X 94.1075,Y 46.6472,Z 105,A 21.37,B 24.9309,C -1.9193,E1 25.1438,E2 424.2142} C_DIS
LIN {X 95.1245,Y 44.5372,Z 105,A 19.4287,B 24.9332,C -1.8881,E1 25.1461,E2 426.2186} C_DIS
LIN {X 96.8915,Y 40.5498,Z 105,A 17.8172,B 24.9314,C -1.9132,E1 25.1478,E2 427.7621} C_DIS
LIN {X 98.5231,Y 36.4084,Z 105,A 15.0286,B 24.933,C -1.8909,E1 25.1506,E2 430.5877} C_DIS
LIN {X 100.375,Y 30.9367,Z 105,A 12.1373,B 24.9329,C -1.8924,E1 25.1531,E2 433.4593} C_DIS
LIN {X 101.354,Y 27.5607,Z 105,A 10.4212,B 24.9327,C -1.895,E1 25.1544,E2 435.1594} C_DIS
LIN {X 102.1939,Y 24.2695,Z 105,A 8.3825,B 24.9336,C -1.8814,E1 25.1558,E2 437.2183} C_DIS
LIN {X 102.9314,Y 20.9131,Z 105,A 6.4978,B 24.9341,C -1.8752,E1 25.1569,E2 439.1068} C_DIS
LIN {X 103.7024,Y 16.6859,Z 105,A 4.2943,B 24.9341,C -1.8737,E1 25.1579,E2 441.3009} C_DIS
LIN {X 104.1534,Y 13.5742,Z 105,A 2.5361,B 24.9347,C -1.8664,E1 25.1586,E2 443.0658} C_DIS
LIN {X 104.8034,Y 6.96,Z 105,A -1.5936,B 24.937,C -1.8336,E1 25.1596,E2 447.2484} C_DIS
LIN {X 104.9881,Y 3.1125,Z 105,A -3.3412,B 24.9364,C -1.8417,E1 25.1598,E2 448.9665} C_DIS
LIN {X 104.9998,Y -2.717,Z 105,A -6.373,B 24.9367,C -1.8377,E1 25.1597,E2 451.9899} C_DIS
LIN {X 104.6516,Y -8.9774,Z 105,A -9.799,B 24.9375,C -1.8263,E1 25.1591,E2 455.4222} C_DIS
LIN {X 104.154,Y -13.5693,Z 105,A -12.5674,B 24.9388,C -1.8077,E1 25.1581,E2 458.2182} C_DIS
LIN {X 103.6886,Y -16.765,Z 105,A -14.1504,B 24.9386,C -1.8095,E1 25.1574,E2 459.7876} C_DIS
LIN {X 102.886,Y -21.1342,Z 105,A -16.9189,B 24.9401,C -1.7872,E1 25.1559,E2 462.5925} C_DIS
LIN {X 102.0167,Y -24.9957,Z 105,A -18.484,B 24.9389,C -1.8053,E1 25.1549,E2 464.1058} C_DIS
LIN {X 101.0528,Y -28.6445,Z 105,A -20.5502,B 24.9394,C -1.7985,E1 25.1534,E2 466.1763} C_DIS
LIN {X 100.0457,Y -31.9872,Z 105,A -22.8276,B 24.9408,C -1.7767,E1 25.1515,E2 468.4921} C_DIS
LIN {X 99.0076,Y -35.0681,Z 105,A -24.1903,B 24.94,C -1.7885,E1 25.1503,E2 469.8193} C_DIS
LIN {X 96.5431,Y -41.3757,Z 105,A -27.7353,B 24.9404,C -1.7834,E1 25.1466,E2 473.3569} C_DIS
LIN {X 94.341,Y -46.1761,Z 105,A -30.9345,B 24.9419,C -1.7612,E1 25.1428,E2 476.5911} C_DIS
LIN {X 91.9423,Y -50.7841,Z 105,A -33.5452,B 24.9418,C -1.7622,E1 25.1394,E2 479.1857} C_DIS
LIN {X 90.5351,Y -53.2507,Z 105,A -35.1035,B 24.9421,C -1.7573,E1 25.1372,E2 480.7475} C_DIS
LIN {X 88.5787,Y -56.4457,Z 105,A -37.1448,B 24.9425,C -1.7516,E1 25.1341,E2 482.7919} C_DIS
LIN {X 86.5805,Y -59.4672,Z 105,A -39.1157,B 24.9429,C -1.7462,E1 25.1311,E2 484.7658} C_DIS
LIN {X 82.2948,Y -65.267,Z 105,A -43.1352,B 24.9438,C -1.732,E1 25.1243,E2 488.7997} C_DIS
LIN {X 80.2705,Y -67.7427,Z 105,A -45.5941,B 24.946,C -1.6977,E1 25.1198,E2 491.3282} C_DIS
LIN {X 76.8372,Y -71.6133,Z 105,A -47.872,B 24.945,C -1.7131,E1 25.1155,E2 493.5599} C_DIS
LIN {X 72.5321,Y -75.9705,Z 105,A -51.4447,B 24.9461,C -1.6954,E1 25.1083,E2 497.1594} C_DIS
LIN {X 69.5779,Y -78.6842,Z 105,A -52.8766,B 24.9445,C -1.7216,E1 25.1055,E2 498.5235} C_DIS
LIN {X 64.6593,Y -82.7751,Z 105,A -56.4043,B 24.9451,C -1.7122,E1 25.0979,E2 502.0601} C_DIS
LIN {X 62.5458,Y -84.3823,Z 105,A -58.6197,B 24.9473,C -1.6776,E1 25.0927,E2 504.3493} C_DIS
LIN {X 59.0039,Y -86.895,Z 105,A -60.4377,B 24.9461,C -1.6954,E1 25.0887,E2 506.1191} C_DIS
LIN {X 55.6881,Y -89.0563,Z 105,A -62.4123,B 24.9459,C -1.6988,E1 25.084,E2 508.0792} C_DIS
LIN {X 52.6715,Y -90.8738,Z 105,A -64.4039,B 24.9463,C -1.6923,E1 25.0792,E2 510.08} C_DIS
LIN {X 49.7842,Y -92.4869,Z 105,A -66.0994,B 24.9463,C -1.6936,E1 25.0751,E2 511.7675} C_DIS
LIN {X 46.6277,Y -94.1172,Z 105,A -68.0889,B 24.9466,C -1.6883,E1 25.0701,E2 513.7641} C_DIS
LIN {X 43.3433,Y -95.6744,Z 105,A -71.1342,B 24.9495,C -1.6423,E1 25.0621,E2 516.9106} C_DIS
LIN {X 37.8217,Y -97.9903,Z 105,A -73.2321,B 24.9468,C -1.6847,E1 25.057,E2 518.9035} C_DIS
LIN {X 30.8006,Y -100.4172,Z 105,A -77.2731,B 24.9471,C -1.68,E1 25.0463,E2 522.9477} C_DIS
LIN {X 26.6051,Y -101.6099,Z 105,A -79.7506,B 24.9475,C -1.6735,E1 25.0396,E2 525.4367} C_DIS
LIN {X 23.5018,Y -102.3712,Z 105,A -81.5398,B 24.9477,C -1.6699,E1 25.0347,E2 527.2317} C_DIS
LIN {X 19.9322,Y -103.1256,Z 105,A -83.6065,B 24.948,C -1.6651,E1 25.029,E2 529.3072} C_DIS
LIN {X 16.0944,Y -103.7938,Z 105,A -85.5949,B 24.9478,C -1.669,E1 25.0236,E2 531.2845} C_DIS
LIN {X 11.8553,Y -104.3636,Z 105,A -88.1904,B 24.9485,C -1.6571,E1 25.0163,E2 533.9062} C_DIS
LIN {X 6.7895,Y -104.815,Z 105,A -90.6235,B 24.9478,C -1.6693,E1 25.0096,E2 536.3092} C_DIS
LIN {X 2.8812,Y -104.9948,Z 105,A -92.9197,B 24.9482,C -1.6621,E1 25.0032,E2 538.6217} C_DIS
LIN {X 2.8812,Y -104.9948,Z 105,A -92.9197,B 24.9482,C -1.6621,E1 25.0032,E2 538.6217} C_DIS
Enddeposition()
LIN {X 0.7307,Y -104.0383,Z 105,A -94.2668,B 24.9476,C -1.6726,E1 24.9995,E2 539.9438} C_DIS
Startdeposition()
$VEL.CP = VEL_PRINT
LIN {X 4.9081,Y -103.9387,Z 105,A -91.1405,B 24.9455,C -1.7053,E1 25.0084,E2 536.7405} C_DIS
LIN {X 8.7965,Y -103.6823,Z 105,A -88.3066,B 24.9437,C -1.7338,E1 25.0165,E2 533.8406} C_DIS
LIN {X 12.1519,Y -103.3416,Z 105,A -86.9888,B 24.945,C -1.7133,E1 25.02,E2 532.5723} C_DIS
LIN {X 15.097,Y -102.9536,Z 105,A -85.2419,B 24.9446,C -1.7188,E1 25.0249,E2 530.8137} C_DIS
LIN {X 18.7733,Y -102.3467,Z 105,A -83.0205,B 24.9441,C -1.7273,E1 25.031,E2 528.5748} C_DIS
LIN {X 22.3218,Y -101.6313,Z 105,A -81.2779,B 24.9446,C -1.719,E1 25.0357,E2 526.8541} C_DIS
LIN {X 25.7487,Y -100.8175,Z 105,A -78.4966,B 24.9423,C -1.7552,E1 25.0435,E2 523.9912} C_DIS
LIN {X 30.4348,Y -99.5039,Z 105,A -76.838,B 24.9448,C -1.7166,E1 25.0477,E2 522.4268} C_DIS
LIN {X 34.4551,Y -98.1835,Z 105,A -74.0009,B 24.9433,C -1.7401,E1 25.0553,E2 519.5396} C_DIS
LIN {X 39.0336,Y -96.455,Z 105,A -70.8629,B 24.9418,C -1.7622,E1 25.0636,E2 516.3565} C_DIS
LIN {X 43.3581,Y -94.5917,Z 105,A -69.1365,B 24.9439,C -1.7304,E1 25.0678,E2 514.7095} C_DIS
LIN {X 46.6732,Y -93.0001,Z 105,A -66.7988,B 24.9428,C -1.7466,E1 25.0737,E2 512.3398} C_DIS
LIN {X 49.4747,Y -91.5392,Z 105,A -65.26,B 24.9432,C -1.7413,E1 25.0774,E2 510.8178} C_DIS
LIN {X 52.3204,Y -89.9446,Z 105,A -63.4772,B 24.943,C -1.744,E1 25.0818,E2 509.0341} C_DIS
LIN {X 55.1117,Y -88.2601,Z 105,A -61.7298,B 24.943,C -1.7454,E1 25.0859,E2 507.2887} C_DIS
LIN {X 57.7239,Y -86.5759,Z 105,A -58.9221,B 24.9396,C -1.7946,E1 25.0927,E2 504.3742} C_DIS
LIN {X 62.5271,Y -83.1716,Z 105,A -56.7824,B 24.9423,C -1.7552,E1 25.0973,E2 502.3352} C_DIS
LIN {X 65.3844,Y -80.9448,Z 105,A -54.1955,B 24.9403,C -1.7844,E1 25.103,E2 499.6892} C_DIS
LIN {X 68.4371,Y -78.3805,Z 105,A -51.9501,B 24.9398,C -1.7915,E1 25.1078,E2 497.4356} C_DIS
LIN {X 71.6048,Y -75.499,Z 105,A -50.4199,B 24.9418,C -1.7623,E1 25.1107,E2 495.9807} C_DIS
LIN {X 73.3307,Y -73.823,Z 105,A -48.1763,B 24.939,C -1.8043,E1 25.1153,E2 493.6476} C_DIS
LIN {X 76.5652,Y -70.4624,Z 105,A -45.8179,B 24.9391,C -1.8018,E1 25.1198,E2 491.3053} C_DIS
LIN {X 79.1452,Y -67.5514,Z 105,A -44.2815,B 24.9405,C -1.7818,E1 25.1225,E2 489.823} C_DIS
LIN {X 81.3209,Y -64.9178,Z 105,A -41.3789,B 24.9372,C -1.8302,E1 25.1277,E2 486.8199} C_DIS
LIN {X 84.6956,Y -60.4467,Z 105,A -39.3724,B 24.9398,C -1.7928,E1 25.1308,E2 484.9113} C_DIS
LIN {X 86.519,Y -57.8102,Z 105,A -37.4537,B 24.939,C -1.8042,E1 25.1339,E2 482.9751} C_DIS
LIN {X 88.3817,Y -54.917,Z 105,A -35.6046,B 24.9387,C -1.8077,E1 25.1366,E2 481.1271} C_DIS
LIN {X 90.2407,Y -51.805,Z 105,A -33.7457,B 24.9387,C -1.8077,E1 25.1392,E2 479.2778} C_DIS
LIN {X 92.7611,Y -47.1442,Z 105,A -30.8804,B 24.9383,C -1.8141,E1 25.143,E2 476.4125} C_DIS
LIN {X 94.4147,Y -43.7384,Z 105,A -28.79,B 24.9379,C -1.8206,E1 25.1455,E2 474.318} C_DIS
LIN {X 95.7955,Y -40.6254,Z 105,A -26.4785,B 24.9362,C -1.8449,E1 25.1481,E2 471.9618} C_DIS
LIN {X 97.6961,Y -35.8141,Z 105,A -24.3558,B 24.9377,C -1.8229,E1 25.1502,E2 469.9028} C_DIS
LIN {X 99.3607,Y -30.8966,Z 105,A -21.282,B 24.9365,C -1.8409,E1 25.1529,E2 466.8039} C_DIS
LIN {X 100.1587,Y -28.203,Z 105,A -19.5787,B 24.9357,C -1.8525,E1 25.1542,E2 465.0831} C_DIS
LIN {X 101.9239,Y -20.9444,Z 105,A -15.7211,B 24.9355,C -1.8547,E1 25.1567,E2 461.2427} C_DIS
LIN {X 102.4881,Y -17.9868,Z 105,A -12.8781,B 24.9316,C -1.9108,E1 25.1581,E2 458.284} C_DIS
LIN {X 103.3287,Y -12.2618,Z 105,A -10.8118,B 24.9342,C -1.873,E1 25.1588,E2 456.319} C_DIS
LIN {X 103.6422,Y -9.249,Z 105,A -9.1625,B 24.9339,C -1.8776,E1 25.1593,E2 454.6686} C_DIS
LIN {X 103.9699,Y -4.1827,Z 105,A -5.6945,B 24.9312,C -1.9154,E1 25.1598,E2 451.1321} C_DIS
LIN {X 104.0553,Y 0.0435,Z 105,A -4.0257,B 24.9327,C -1.8947,E1 25.1598,E2 449.5219} C_DIS
LIN {X 103.8521,Y 6.4929,Z 105,A -0.631,B 24.9324,C -1.8994,E1 25.1594,E2 446.1364} C_DIS
LIN {X 103.4933,Y 10.7833,Z 105,A 1.8409,B 24.9315,C -1.9113,E1 25.1588,E2 443.6512} C_DIS
LIN {X 103.0988,Y 14.0752,Z 105,A 3.8857,B 24.9304,C -1.9264,E1 25.1581,E2 441.5829} C_DIS
LIN {X 102.4072,Y 18.4368,Z 105,A 6.0908,B 24.9306,C -1.9244,E1 25.157,E2 439.3952} C_DIS
LIN {X 101.7243,Y 21.895,Z 105,A 8.0253,B 24.9302,C -1.9302,E1 25.1559,E2 437.4584} C_DIS
LIN {X 100.9936,Y 25.0518,Z 105,A 9.9865,B 24.9292,C -1.9432,E1 25.1546,E2 435.4779} C_DIS
LIN {X 100.0541,Y 28.5721,Z 105,A 11.7752,B 24.9294,C -1.9402,E1 25.1533,E2 433.7066} C_DIS
LIN {X 98.2644,Y 34.2245,Z 105,A 15.0979,B 24.9285,C -1.9524,E1 25.1504,E2 430.3738} C_DIS
LIN {X 96.4617,Y 39.0172,Z 105,A 17.8619,B 24.9281,C -1.9583,E1 25.1477,E2 427.6112} C_DIS
LIN {X 94.2051,Y 44.1887,Z 105,A 20.7007,B 24.9283,C -1.956,E1 25.1445,E2 424.7935} C_DIS
LIN {X 93.18,Y 46.3104,Z 105,A 22.2029,B 24.9274,C -1.9682,E1 25.1426,E2 423.2704} C_DIS
LIN {X 91.4431,Y 49.6518,Z 105,A 24.9198,B 24.9249,C -2.001,E1 25.1389,E2 420.4904} C_DIS
LIN {X 89.3367,Y 53.3509,Z 105,A 26.5147,B 24.9268,C -1.9758,E1 25.1368,E2 418.9633} C_DIS
LIN {X 87.731,Y 55.9509,Z 105,A 28.7086,B 24.9249,C -2.0016,E1 25.1334,E2 416.7195} C_DIS
LIN {X 85.8529,Y 58.794,Z 105,A 29.9982,B 24.9264,C -1.9818,E1 25.1315,E2 415.4829} C_DIS
LIN {X 83.6953,Y 61.8259,Z 105,A 32.6347,B 24.9241,C -2.0114,E1 25.127,E2 412.7892} C_DIS
LIN {X 81.6449,Y 64.5079,Z 105,A 33.6306,B 24.9265,C -1.9801,E1 25.1255,E2 411.8719} C_DIS
LIN {X 79.2196,Y 67.4641,Z 105,A 36.0716,B 24.9251,C -1.9989,E1 25.1211,E2 409.3979} C_DIS
LIN {X 77.0668,Y 69.9157,Z 105,A 38.68,B 24.9222,C -2.0366,E1 25.116,E2 406.7119} C_DIS
LIN {X 73.8897,Y 73.2632,Z 105,A 40.4409,B 24.9243,C -2.0098,E1 25.1127,E2 405.0219} C_DIS
LIN {X 68.3034,Y 78.4973,Z 105,A 44.6792,B 24.9235,C -2.0193,E1 25.104,E2 400.7785} C_DIS
LIN {X 66.2048,Y 80.276,Z 105,A 46.4399,B 24.9226,C -2.0322,E1 25.1002,E2 398.9939} C_DIS
LIN {X 62.0067,Y 83.5625,Z 105,A 48.9733,B 24.9234,C -2.0211,E1 25.0946,E2 396.4961} C_DIS
LIN {X 56.3171,Y 87.496,Z 105,A 52.8344,B 24.9228,C -2.0294,E1 25.0857,E2 392.6282} C_DIS
LIN {X 53.473,Y 89.2646,Z 105,A 54.8606,B 24.922,C -2.0396,E1 25.0808,E2 390.5844} C_DIS
LIN {X 50.6501,Y 90.894,Z 105,A 56.4246,B 24.9225,C -2.0328,E1 25.0771,E2 389.041} C_DIS
LIN {X 47.4697,Y 92.5948,Z 105,A 58.1349,B 24.9232,C -2.0244,E1 25.0729,E2 387.3554} C_DIS
LIN {X 45.126,Y 93.7593,Z 105,A 60.61,B 24.9198,C -2.0678,E1 25.0665,E2 384.7842} C_DIS
LIN {X 41.0665,Y 95.6086,Z 105,A 62.3291,B 24.9219,C -2.0408,E1 25.0622,E2 383.1331} C_DIS
LIN {X 38.033,Y 96.8537,Z 105,A 64.1919,B 24.9216,C -2.045,E1 25.0574,E2 381.2648} C_DIS
LIN {X 33.9545,Y 98.3588,Z 105,A 66.7668,B 24.9209,C -2.0543,E1 25.0506,E2 378.673} C_DIS
LIN {X 30.7768,Y 99.3979,Z 105,A 68.3759,B 24.9215,C -2.0466,E1 25.0464,E2 377.0851} C_DIS
LIN {X 24.7976,Y 101.0557,Z 105,A 71.5542,B 24.922,C -2.0394,E1 25.0379,E2 373.9289} C_DIS
LIN {X 21.3004,Y 101.8508,Z 105,A 73.5626,B 24.9218,C -2.0417,E1 25.0324,E2 371.9178} C_DIS
LIN {X 17.389,Y 102.5906,Z 105,A 75.9727,B 24.9211,C -2.0511,E1 25.0257,E2 369.4882} C_DIS
LIN {X 14.2001,Y 103.081,Z 105,A 77.8189,B 24.9209,C -2.0542,E1 25.0206,E2 367.6361} C_DIS
LIN {X 10.7271,Y 103.4992,Z 105,A 79.6637,B 24.9211,C -2.0514,E1 25.0155,E2 365.7993} C_DIS
LIN {X 7.7702,Y 103.7644,Z 105,A 81.1994,B 24.9214,C -2.0477,E1 25.0112,E2 364.2733} C_DIS
LIN {X 3.4103,Y 103.9979,Z 105,A 83.6013,B 24.9214,C -2.0475,E1 25.0045,E2 361.8726} C_DIS
LIN {X 0.4441,Y 104.0528,Z 105,A 85.3627,B 24.921,C -2.0521,E1 24.9996,E2 360.1004} C_DIS
LIN {X -6.3586,Y 103.861,Z 105,A 88.9954,B 24.9215,C -2.0465,E1 24.9895,E2 356.4804} C_DIS
LIN {X -10.5722,Y 103.5154,Z 105,A 91.4676,B 24.9211,C -2.0509,E1 24.9826,E2 353.9965} C_DIS
LIN {X -13.7948,Y 103.136,Z 105,A 93.2788,B 24.9211,C -2.0507,E1 24.9776,E2 352.1844} C_DIS
LIN {X -17.3633,Y 102.5949,Z 105,A 95.1607,B 24.9216,C -2.0454,E1 24.9724,E2 350.3135} C_DIS
LIN {X -22.904,Y 101.5029,Z 105,A 99.0186,B 24.9196,C -2.0711,E1 24.9617,E2 346.3899} C_DIS
LIN {X -27.1011,Y 100.4623,Z 105,A 100.6989,B 24.9218,C -2.0422,E1 24.9573,E2 344.7759} C_DIS
LIN {X -34.188,Y 98.2772,Z 105,A 104.5326,B 24.9229,C -2.028,E1 24.9472,E2 340.969} C_DIS
LIN {X -38.5297,Y 96.6586,Z 105,A 107.2579,B 24.9226,C -2.031,E1 24.9401,E2 338.2308} C_DIS
LIN {X -41.1444,Y 95.5747,Z 105,A 109.3839,B 24.9212,C -2.0499,E1 24.9344,E2 336.0549} C_DIS
LIN {X -44.2621,Y 94.1709,Z 105,A 111.116,B 24.9219,C -2.0414,E1 24.9301,E2 334.3388} C_DIS
LIN {X -48.6617,Y 91.9741,Z 105,A 113.5793,B 24.9229,C -2.0279,E1 24.9241,E2 331.9009} C_DIS
LIN {X -56.3895,Y 87.4495,Z 105,A 118.5811,B 24.9234,C -2.0214,E1 24.9121,E2 326.8993} C_DIS
LIN {X -59.617,Y 85.2821,Z 105,A 120.5594,B 24.9242,C -2.0112,E1 24.9076,E2 324.9387} C_DIS
LIN {X -62.1899,Y 83.4249,Z 105,A 122.4577,B 24.924,C -2.0131,E1 24.9033,E2 323.0292} C_DIS
LIN {X -65.0212,Y 81.2391,Z 105,A 124.477,B 24.9242,C -2.0106,E1 24.8988,E2 321.0082} C_DIS
LIN {X -67.6618,Y 79.0512,Z 105,A 126.2221,B 24.9249,C -2.0012,E1 24.8951,E2 319.2787} C_DIS
LIN {X -70.3238,Y 76.6924,Z 105,A 128.2068,B 24.9252,C -1.9977,E1 24.891,E2 317.2946} C_DIS
LIN {X -72.8888,Y 74.2596,Z 105,A 130.2115,B 24.9254,C -1.9951,E1 24.887,E2 315.2876} C_DIS
LIN {X -75.3775,Y 71.734,Z 105,A 132.2676,B 24.9254,C -1.9941,E1 24.883,E2 313.2252} C_DIS
LIN {X -77.7118,Y 69.1961,Z 105,A 134.1067,B 24.926,C -1.9871,E1 24.8795,E2 311.3945} C_DIS
LIN {X -80.0144,Y 66.5195,Z 105,A 136.0324,B 24.9264,C -1.9814,E1 24.8761,E2 309.4735} C_DIS
LIN {X -82.4701,Y 63.4494,Z 105,A 138.1137,B 24.927,C -1.9727,E1 24.8725,E2 307.4033} C_DIS
LIN {X -84.3796,Y 60.8896,Z 105,A 140.0467,B 24.927,C -1.9741,E1 24.8693,E2 305.4574} C_DIS
LIN {X -87.4275,Y 56.4238,Z 105,A 142.9669,B 24.9277,C -1.9638,E1 24.8648,E2 302.5474} C_DIS
LIN {X -90.5332,Y 51.2945,Z 105,A 146.1733,B 24.9286,C -1.9508,E1 24.8602,E2 299.3553} C_DIS
LIN {X -92.6867,Y 47.2899,Z 105,A 149.2071,B 24.9278,C -1.9624,E1 24.8562,E2 296.2777} C_DIS
LIN {X -94.1343,Y 44.3408,Z 105,A 150.4522,B 24.9297,C -1.9368,E1 24.8548,E2 295.0868} C_DIS
LIN {X -95.836,Y 40.5294,Z 105,A 152.5914,B 24.9306,C -1.9242,E1 24.8524,E2 292.966} C_DIS
LIN {X -97.3049,Y 36.8634,Z 105,A 154.7205,B 24.9312,C -1.9159,E1 24.8502,E2 290.8449} C_DIS
LIN {X -99.1084,Y 31.6986,Z 105,A 157.8833,B 24.9315,C -1.9117,E1 24.8473,E2 287.674} C_DIS
LIN {X -99.802,Y 29.4403,Z 105,A 159.4329,B 24.9311,C -1.9165,E1 24.846,E2 286.1042} C_DIS
LIN {X -100.733,Y 26.0777,Z 105,A 161.2968,B 24.9317,C -1.9083,E1 24.8447,E2 284.2488} C_DIS
LIN {X -101.5673,Y 22.6147,Z 105,A 163.2321,B 24.9322,C -1.9011,E1 24.8434,E2 282.3193} C_DIS
LIN {X -102.1574,Y 19.7745,Z 105,A 164.9668,B 24.9322,C -1.9009,E1 24.8425,E2 280.575} C_DIS
LIN {X -102.7076,Y 16.6891,Z 105,A 167.6345,B 24.9302,C -1.929,E1 24.8413,E2 277.8242} C_DIS
LIN {X -103.4167,Y 11.5106,Z 105,A 169.5332,B 24.9334,C -1.8847,E1 24.8407,E2 276.0201} C_DIS
LIN {X -103.71,Y 8.4503,Z 105,A 171.3175,B 24.9336,C -1.8825,E1 24.8402,E2 274.2302} C_DIS
LIN {X -103.9232,Y 5.2317,Z 105,A 173.2232,B 24.9336,C -1.8813,E1 24.8399,E2 272.3159} C_DIS
LIN {X -104.0399,Y 1.7038,Z 105,A 175.0414,B 24.9344,C -1.8706,E1 24.8398,E2 270.5123} C_DIS
LIN {X -104.0372,Y -1.8476,Z 105,A 177.0809,B 24.9346,C -1.8673,E1 24.8398,E2 268.4685} C_DIS
LIN {X -103.9055,Y -5.5531,Z 105,A 179.1241,B 24.9351,C -1.8608,E1 24.8401,E2 266.4285} C_DIS
LIN {X -103.6499,Y -9.1651,Z 105,A -178.8573,B 24.9355,C -1.8553,E1 24.8405,E2 264.4109} C_DIS
LIN {X -103.285,Y -12.6349,Z 105,A -176.8475,B 24.9357,C -1.8523,E1 24.8412,E2 262.3961} C_DIS
LIN {X -102.7943,Y -16.1413,Z 105,A -175.0281,B 24.9364,C -1.8415,E1 24.8419,E2 260.5916} C_DIS
LIN {X -101.8316,Y -21.3939,Z 105,A -172.2997,B 24.9376,C -1.8247,E1 24.8433,E2 257.887} C_DIS
LIN {X -100.8393,Y -25.6643,Z 105,A -169.5898,B 24.9374,C -1.8278,E1 24.8451,E2 255.1539} C_DIS
LIN {X -99.9445,Y -28.9588,Z 105,A -166.5275,B 24.9348,C -1.8649,E1 24.8476,E2 251.9856} C_DIS
LIN {X -98.0205,Y -34.9197,Z 105,A -164.2147,B 24.9384,C -1.8133,E1 24.8496,E2 249.7826} C_DIS
LIN {X -96.8566,Y -38.0255,Z 105,A -162.3856,B 24.9387,C -1.8081,E1 24.8514,E2 247.9557} C_DIS
LIN {X -95.5035,Y -41.3076,Z 105,A -160.3877,B 24.939,C -1.804,E1 24.8536,E2 245.9565} C_DIS
LIN {X -94.0164,Y -44.5908,Z 105,A -157.8986,B 24.9381,C -1.8166,E1 24.8566,E2 243.4237} C_DIS
LIN {X -92.3453,Y -47.9569,Z 105,A -156.4605,B 24.9401,C -1.788,E1 24.8584,E2 242.0461} C_DIS
LIN {X -90.4186,Y -51.4955,Z 105,A -154.3291,B 24.9407,C -1.7788,E1 24.8612,E2 239.9255} C_DIS
LIN {X -88.5559,Y -54.6382,Z 105,A -152.0184,B 24.9403,C -1.7843,E1 24.8646,E2 237.5898} C_DIS
LIN {X -86.7363,Y -57.4807,Z 105,A -150.1477,B 24.9406,C -1.7799,E1 24.8674,E2 235.72} C_DIS
LIN {X -83.9365,Y -61.4965,Z 105,A -147.5088,B 24.9412,C -1.7711,E1 24.8717,E2 233.0892} C_DIS
LIN {X -81.4362,Y -64.7718,Z 105,A -145.3236,B 24.9418,C -1.7626,E1 24.8754,E2 230.914} C_DIS
LIN {X -79.4462,Y -67.1981,Z 105,A -142.5611,B 24.9395,C -1.7968,E1 24.8806,E2 228.0573} C_DIS
LIN {X -75.9135,Y -71.164,Z 105,A -140.8873,B 24.943,C -1.744,E1 24.8835,E2 226.5019} C_DIS
LIN {X -74.1816,Y -72.9678,Z 105,A -138.5946,B 24.941,C -1.7749,E1 24.8881,E2 224.1259} C_DIS
LIN {X -71.3822,Y -75.7083,Z 105,A -137.0211,B 24.9427,C -1.7487,E1 24.8912,E2 222.6082} C_DIS
LIN {X -68.7694,Y -78.0903,Z 105,A -134.773,B 24.9422,C -1.756,E1 24.8959,E2 220.3337} C_DIS
LIN {X -65.8939,Y -80.5318,Z 105,A -132.8229,B 24.9428,C -1.7473,E1 24.9001,E2 218.3968} C_DIS
LIN {X -62.9403,Y -82.8612,Z 105,A -130.1726,B 24.9416,C -1.7654,E1 24.9061,E2 215.6939} C_DIS
LIN {X -59.3895,Y -85.4402,Z 105,A -128.7387,B 24.9443,C -1.7244,E1 24.9092,E2 214.3526} C_DIS
LIN {X -57.2387,Y -86.8958,Z 105,A -127.0277,B 24.9437,C -1.7326,E1 24.9132,E2 212.6164} C_DIS
LIN {X -53.5561,Y -89.2145,Z 105,A -124.7158,B 24.9442,C -1.7258,E1 24.9187,E2 210.3134} C_DIS
LIN {X -50.2102,Y -91.1397,Z 105,A -122.5948,B 24.9444,C -1.7227,E1 24.9238,E2 208.1937} C_DIS
LIN {X -44.1393,Y -94.2281,Z 105,A -118.6958,B 24.9444,C -1.7236,E1 24.9336,E2 204.282} C_DIS
LIN {X -40.949,Y -95.6592,Z 105,A -116.6896,B 24.9443,C -1.7246,E1 24.9387,E2 202.2689} C_DIS
LIN {X -36.8977,Y -97.2919,Z 105,A -114.187,B 24.9442,C -1.7261,E1 24.9453,E2 199.7574} C_DIS
LIN {X -34.1429,Y -98.293,Z 105,A -112.6825,B 24.9445,C -1.7205,E1 24.9492,E2 198.2633} C_DIS
LIN {X -27.9733,Y -100.2238,Z 105,A -109.3362,B 24.9452,C -1.7096,E1 24.9581,E2 194.937} C_DIS
LIN {X -24.7289,Y -101.0724,Z 105,A -107.5177,B 24.9454,C -1.7075,E1 24.963,E2 193.121} C_DIS
LIN {X -22.1043,Y -101.6787,Z 105,A -105.9012,B 24.9451,C -1.7119,E1 24.9674,E2 191.4919} C_DIS
LIN {X -18.5434,Y -102.388,Z 105,A -103.8583,B 24.9451,C -1.7129,E1 24.9731,E2 189.4445} C_DIS
LIN {X -15.0147,Y -102.9653,Z 105,A -101.8655,B 24.945,C -1.7133,E1 24.9786,E2 187.449} C_DIS
LIN {X -10.6637,Y -103.5058,Z 105,A -99.6778,B 24.9456,C -1.704,E1 24.9846,E2 185.2817} C_DIS
LIN {X -5.8429,Y -103.8895,Z 105,A -96.855,B 24.9452,C -1.7103,E1 24.9925,E2 182.443} C_DIS
LIN {X -2.6905,Y -104.02,Z 105,A -94.4221,B 24.9434,C -1.7381,E1 24.9995,E2 179.9438} C_DIS
LIN {X 0.7307,Y -104.0383,Z 105,A -94.2624,B 24.9477,C -1.6708,E1 24.9995,E2 179.9438} C_DIS
Enddeposition()
LIN {X 0.7307,Y -104.0383,Z 105,A -94.2624,B 24.9477,C -1.6708,E1 24.9995,E2 179.9438} C_DIS
Startdeposition()
$VEL.CP = VEL_PRINT
LIN {X -0.4969,Y -103.0719,Z 105,A -94.7737,B 24.9462,C -1.6943,E1 24.9982,E2 180.3992} C_DIS
LIN {X -4.3036,Y -102.9832,Z 105,A -96.8781,B 24.9462,C -1.6945,E1 24.9923,E2 182.5035} C_DIS
LIN {X -9.1327,Y -102.6681,Z 105,A -99.4669,B 24.9459,C -1.6984,E1 24.9851,E2 185.0841} C_DIS
LIN {X -12.6103,Y -102.3006,Z 105,A -101.5961,B 24.9464,C -1.6916,E1 24.9792,E2 187.2309} C_DIS
LIN {X -16.0373,Y -101.8181,Z 105,A -103.4957,B 24.9463,C -1.693,E1 24.9739,E2 189.1287} C_DIS
LIN {X -19.4777,Y -101.2159,Z 105,A -105.3445,B 24.946,C -1.6972,E1 24.9689,E2 190.9695} C_DIS
LIN {X -22.9187,Y -100.4931,Z 105,A -107.0919,B 24.9455,C -1.7059,E1 24.9642,E2 192.6983} C_DIS
LIN {X -25.2321,Y -99.9378,Z 105,A -108.7832,B 24.9463,C -1.6927,E1 24.9595,E2 194.4232} C_DIS
LIN {X -31.5249,Y -98.1339,Z 105,A -112.1931,B 24.9456,C -1.7038,E1 24.9504,E2 197.8125} C_DIS
LIN {X -35.8383,Y -96.6431,Z 105,A -114.9415,B 24.946,C -1.6981,E1 24.9431,E2 200.5799} C_DIS
LIN {X -39.3495,Y -95.2677,Z 105,A -117.0205,B 24.9458,C -1.7008,E1 24.9377,E2 202.657} C_DIS
LIN {X -42.5103,Y -93.8986,Z 105,A -118.8044,B 24.9453,C -1.7078,E1 24.9332,E2 204.4286} C_DIS
LIN {X -44.6657,Y -92.8925,Z 105,A -120.5593,B 24.9463,C -1.6934,E1 24.9287,E2 206.2222} C_DIS
LIN {X -47.5474,Y -91.4526,Z 105,A -122.0658,B 24.9454,C -1.7061,E1 24.925,E2 207.7026} C_DIS
LIN {X -51.9642,Y -89.0173,Z 105,A -125.0197,B 24.9456,C -1.7045,E1 24.9178,E2 210.669} C_DIS
LIN {X -55.5145,Y -86.846,Z 105,A -127.107,B 24.9448,C -1.7163,E1 24.9129,E2 212.7349} C_DIS
LIN {X -58.4425,Y -84.9043,Z 105,A -129.1035,B 24.9447,C -1.7179,E1 24.9083,E2 214.7343} C_DIS
LIN {X -62.3338,Y -82.0903,Z 105,A -131.897,B 24.9447,C -1.7179,E1 24.902,E2 217.5373} C_DIS
LIN {X -65.4958,Y -79.5901,Z 105,A -133.9168,B 24.9439,C -1.7301,E1 24.8977,E2 219.5359} C_DIS
LIN {X -68.2785,Y -77.2171,Z 105,A -136.1297,B 24.9441,C -1.7276,E1 24.8929,E2 221.7635} C_DIS
LIN {X -70.3445,Y -75.3381,Z 105,A -137.9082,B 24.9444,C -1.7226,E1 24.8893,E2 223.561} C_DIS
LIN {X -73.6357,Y -72.125,Z 105,A -140.2381,B 24.9435,C -1.7362,E1 24.8847,E2 225.8685} C_DIS
LIN {X -75.9846,Y -69.6446,Z 105,A -142.6568,B 24.9444,C -1.7219,E1 24.8801,E2 228.3318} C_DIS
LIN {X -78.5765,Y -66.7069,Z 105,A -144.3389,B 24.943,C -1.7445,E1 24.8771,E2 229.9678} C_DIS
LIN {X -80.6018,Y -64.2462,Z 105,A -146.1082,B 24.9427,C -1.7488,E1 24.874,E2 231.7352} C_DIS
LIN {X -83.7989,Y -60.0152,Z 105,A -149.1738,B 24.9425,C -1.7519,E1 24.8689,E2 234.8082} C_DIS
LIN {X -86.081,Y -56.6931,Z 105,A -151.2658,B 24.9418,C -1.7628,E1 24.8656,E2 236.8845} C_DIS
LIN {X -87.9421,Y -53.7614,Z 105,A -153.2185,B 24.9415,C -1.7671,E1 24.8627,E2 238.8369} C_DIS
LIN {X -89.7428,Y -50.7004,Z 105,A -155.5348,B 24.9419,C -1.7604,E1 24.8595,E2 241.1814} C_DIS
LIN {X -91.8971,Y -46.68,Z 105,A -158.1342,B 24.9416,C -1.7652,E1 24.8562,E2 243.7832} C_DIS
LIN {X -93.9644,Y -42.3643,Z 105,A -160.4283,B 24.9402,C -1.7855,E1 24.8535,E2 246.0414} C_DIS
LIN {X -95.3556,Y -39.1336,Z 105,A -162.395,B 24.9399,C -1.7907,E1 24.8514,E2 248.0066} C_DIS
LIN {X -96.5589,Y -36.0644,Z 105,A -164.2949,B 24.9397,C -1.7937,E1 24.8495,E2 249.9099} C_DIS
LIN {X -98.5406,Y -30.2304,Z 105,A -167.6621,B 24.9389,C -1.806,E1 24.8465,E2 253.2671} C_DIS
LIN {X -99.6457,Y -26.3639,Z 105,A -170.5198,B 24.9399,C -1.7913,E1 24.8444,E2 256.1764} C_DIS
LIN {X -100.5659,Y -22.5953,Z 105,A -172.161,B 24.9382,C -1.8158,E1 24.8434,E2 257.769} C_DIS
LIN {X -101.6652,Y -16.9771,Z 105,A -175.3008,B 24.9374,C -1.8272,E1 24.8418,E2 260.9001} C_DIS
LIN {X -102.2033,Y -13.3614,Z 105,A -177.3607,B 24.937,C -1.8327,E1 24.841,E2 262.9593} C_DIS
LIN {X -102.6042,Y -9.825,Z 105,A -179.3582,B 24.9367,C -1.8383,E1 24.8404,E2 264.9553} C_DIS
LIN {X -102.8858,Y -6.2332,Z 105,A 178.5675,B 24.9364,C -1.8422,E1 24.84,E2 267.0326} C_DIS
LIN {X -103.0368,Y -2.7605,Z 105,A 176.609,B 24.936,C -1.8475,E1 24.8398,E2 268.9903} C_DIS
LIN {X -103.07,Y 0.8257,Z 105,A 174.6674,B 24.9354,C -1.8558,E1 24.8398,E2 270.924} C_DIS
LIN {X -102.9755,Y 4.4809,Z 105,A 172.6455,B 24.935,C -1.8627,E1 24.84,E2 272.9415} C_DIS
LIN {X -102.7499,Y 8.1544,Z 105,A 170.5672,B 24.9346,C -1.8682,E1 24.8404,E2 275.0192} C_DIS
LIN {X -102.4869,Y 10.979,Z 105,A 168.4168,B 24.9356,C -1.8536,E1 24.8411,E2 277.2172} C_DIS
LIN {X -102.0055,Y 14.793,Z 105,A 166.4667,B 24.9347,C -1.8669,E1 24.8418,E2 279.1473} C_DIS
LIN {X -101.2067,Y 19.5256,Z 105,A 164.2015,B 24.9331,C -1.8893,E1 24.8429,E2 281.3725} C_DIS
LIN {X -100.4754,Y 22.9949,Z 105,A 162.4699,B 24.932,C -1.9039,E1 24.8439,E2 283.0795} C_DIS
LIN {X -99.8936,Y 25.4042,Z 105,A 160.7662,B 24.9325,C -1.897,E1 24.8451,E2 284.8096} C_DIS
Enddeposition()
END
